   1:L PR[91] 10mm/sec CNT100;
   1:  PR[GP1:91,1] = PR[GP1:90,1] + -19.480;
   1:  PR[GP1:91,2] = PR[GP1:90,2] + 30.902;
   1:L PR[91] 10mm/sec CNT100;
   1:  PR[GP1:91,1] = PR[GP1:90,1] + -27.630;
   1:  PR[GP1:91,2] = PR[GP1:90,2] + 34.001;
   1:L PR[91] 10mm/sec CNT100;
   1:  PR[GP1:91,1] = PR[GP1:90,1] + -29.966;
   1:  PR[GP1:91,2] = PR[GP1:90,2] + 34.343;
   1:L PR[91] 10mm/sec CNT100;
   1:  PR[GP1:91,1] = PR[GP1:90,1] + -37.896;
   1:  PR[GP1:91,2] = PR[GP1:90,2] + 34.907;
   1:L PR[91] 10mm/sec CNT100;
   1:  PR[GP1:91,1] = PR[GP1:90,1] + -42.869;
   1:  PR[GP1:91,2] = PR[GP1:90,2] + 34.106;
   1:L PR[91] 10mm/sec CNT100;
   1:  PR[GP1:91,1] = PR[GP1:90,1] + -48.250;
   1:  PR[GP1:91,2] = PR[GP1:90,2] + 32.901;
   1:L PR[91] 10mm/sec CNT100;
   1:  PR[GP1:91,1] = PR[GP1:90,1] + -54.688;
   1:  PR[GP1:91,2] = PR[GP1:90,2] + 29.663;
   1:L PR[91] 10mm/sec CNT100;
   1:  PR[GP1:91,1] = PR[GP1:90,1] + -57.745;
   1:  PR[GP1:91,2] = PR[GP1:90,2] + 27.940;
   1:L PR[91] 10mm/sec CNT100;
   1:  PR[GP1:91,1] = PR[GP1:90,1] + -63.977;
   1:  PR[GP1:91,2] = PR[GP1:90,2] + 21.826;
   1:L PR[91] 10mm/sec CNT100;
   1:  PR[GP1:91,1] = PR[GP1:90,1] + -65.405;
   1:  PR[GP1:91,2] = PR[GP1:90,2] + 20.322;
   1:L PR[91] 10mm/sec CNT100;
   1:  PR[GP1:91,1] = PR[GP1:90,1] + -69.842;
   1:  PR[GP1:91,2] = PR[GP1:90,2] + 11.800;
   1:L PR[91] 10mm/sec CNT100;
   1:  PR[GP1:91,1] = PR[GP1:90,1] + -70.385;
   1:  PR[GP1:91,2] = PR[GP1:90,2] + 10.702;
   1:L PR[91] 10mm/sec CNT100;
   1:  PR[GP1:91,1] = PR[GP1:90,1] + -71.982;
   1:  PR[GP1:91,2] = PR[GP1:90,2] + 0.854;
   1:L PR[91] 10mm/sec CNT100;
   1:  PR[GP1:91,1] = PR[GP1:90,1] + -72.151;
   1:  PR[GP1:91,2] = PR[GP1:90,2] + -0.013;
   1:L PR[91] 10mm/sec CNT100;
   1:  PR[GP1:91,1] = PR[GP1:90,1] + -70.545;
   1:  PR[GP1:91,2] = PR[GP1:90,2] + -9.656;
   1:L PR[91] 10mm/sec CNT100;
   1:  PR[GP1:91,1] = PR[GP1:90,1] + -70.383;
   1:  PR[GP1:91,2] = PR[GP1:90,2] + -10.713;
   1:L PR[91] 10mm/sec CNT100;
   1:  PR[GP1:91,1] = PR[GP1:90,1] + -69.842;
   1:  PR[GP1:91,2] = PR[GP1:90,2] + -11.809;
   1:L PR[91] 10mm/sec CNT100;
   1:  PR[GP1:91,1] = PR[GP1:90,1] + -65.405;
   1:  PR[GP1:91,2] = PR[GP1:90,2] + -20.330;
   1:L PR[91] 10mm/sec CNT100;
   1:  PR[GP1:91,1] = PR[GP1:90,1] + -63.977;
   1:  PR[GP1:91,2] = PR[GP1:90,2] + -21.835;
   1:L PR[91] 10mm/sec CNT100;
   1:  PR[GP1:91,1] = PR[GP1:90,1] + -57.745;
   1:  PR[GP1:91,2] = PR[GP1:90,2] + -27.949;
   1:L PR[91] 10mm/sec CNT100;
   1:  PR[GP1:91,1] = PR[GP1:90,1] + -54.688;
   1:  PR[GP1:91,2] = PR[GP1:90,2] + -29.672;
   1:L PR[91] 10mm/sec CNT100;
   1:  PR[GP1:91,1] = PR[GP1:90,1] + -48.250;
   1:  PR[GP1:91,2] = PR[GP1:90,2] + -32.910;
   1:L PR[91] 10mm/sec CNT100;
   1:  PR[GP1:91,1] = PR[GP1:90,1] + -42.869;
   1:  PR[GP1:91,2] = PR[GP1:90,2] + -34.115;
   1:L PR[91] 10mm/sec CNT100;
   1:  PR[GP1:91,1] = PR[GP1:90,1] + -37.896;
   1:  PR[GP1:91,2] = PR[GP1:90,2] + -34.916;
   1:L PR[91] 10mm/sec CNT100;
   1:  PR[GP1:91,1] = PR[GP1:90,1] + -29.966;
   1:  PR[GP1:91,2] = PR[GP1:90,2] + -34.352;
   1:L PR[91] 10mm/sec CNT100;
   1:  PR[GP1:91,1] = PR[GP1:90,1] + -27.630;
   1:  PR[GP1:91,2] = PR[GP1:90,2] + -34.009;
   1:L PR[91] 10mm/sec CNT100;
   1:  PR[GP1:91,1] = PR[GP1:90,1] + -19.480;
   1:  PR[GP1:91,2] = PR[GP1:90,2] + -30.911;
   1:L PR[91] 10mm/sec CNT100;
   1:  PR[GP1:91,1] = PR[GP1:90,1] + -18.119;
   1:  PR[GP1:91,2] = PR[GP1:90,2] + -30.431;
   1:L PR[91] 10mm/sec CNT100;
   1:  PR[GP1:91,1] = PR[GP1:90,1] + -17.970;
   1:  PR[GP1:91,2] = PR[GP1:90,2] + -30.350;
   1:L PR[91] 10mm/sec CNT100;
   1:  PR[GP1:91,1] = PR[GP1:90,1] + -10.591;
   1:  PR[GP1:91,2] = PR[GP1:90,2] + -24.946;
   1:L PR[91] 10mm/sec CNT100;
   1:  PR[GP1:91,1] = PR[GP1:90,1] + -9.471;
   1:  PR[GP1:91,2] = PR[GP1:90,2] + -24.053;
   1:L PR[91] 10mm/sec CNT100;
   1:  PR[GP1:91,1] = PR[GP1:90,1] + -8.184;
   1:  PR[GP1:91,2] = PR[GP1:90,2] + -22.548;
   1:L PR[91] 10mm/sec CNT100;
   1:  PR[GP1:91,1] = PR[GP1:90,1] + -4.096;
   1:  PR[GP1:91,2] = PR[GP1:90,2] + -16.957;
   1:L PR[91] 10mm/sec CNT100;
   1:  PR[GP1:91,1] = PR[GP1:90,1] + -2.895;
   1:  PR[GP1:91,2] = PR[GP1:90,2] + -15.610;
   1:L PR[91] 10mm/sec CNT100;
   1:  PR[GP1:91,1] = PR[GP1:90,1] + -0.647;
   1:  PR[GP1:91,2] = PR[GP1:90,2] + -14.295;
   1:L PR[91] 10mm/sec CNT100;
   1:  PR[GP1:91,1] = PR[GP1:90,1] + 1.549;
   1:  PR[GP1:91,2] = PR[GP1:90,2] + -14.273;
   1:L PR[91] 10mm/sec CNT100;
   1:  PR[GP1:91,1] = PR[GP1:90,1] + 2.672;
   1:  PR[GP1:91,2] = PR[GP1:90,2] + -15.619;
   1:L PR[91] 10mm/sec CNT100;
   1:  PR[GP1:91,1] = PR[GP1:90,1] + 3.279;
   1:  PR[GP1:91,2] = PR[GP1:90,2] + -16.002;
   1:L PR[91] 10mm/sec CNT100;
   1:  PR[GP1:91,1] = PR[GP1:90,1] + 4.858;
   1:  PR[GP1:91,2] = PR[GP1:90,2] + -16.866;
   1:L PR[91] 10mm/sec CNT100;
   1:  PR[GP1:91,1] = PR[GP1:90,1] + 9.010;
   1:  PR[GP1:91,2] = PR[GP1:90,2] + -22.547;
   1:L PR[91] 10mm/sec CNT100;
   1:  PR[GP1:91,1] = PR[GP1:90,1] + 10.298;
   1:  PR[GP1:91,2] = PR[GP1:90,2] + -24.056;
   1:L PR[91] 10mm/sec CNT100;
   1:  PR[GP1:91,1] = PR[GP1:90,1] + 18.793;
   1:  PR[GP1:91,2] = PR[GP1:90,2] + -30.355;
   1:L PR[91] 10mm/sec CNT100;
   1:  PR[GP1:91,1] = PR[GP1:90,1] + 18.939;
   1:  PR[GP1:91,2] = PR[GP1:90,2] + -30.434;
   1:L PR[91] 10mm/sec CNT100;
   1:  PR[GP1:91,1] = PR[GP1:90,1] + 20.300;
   1:  PR[GP1:91,2] = PR[GP1:90,2] + -30.914;
   1:L PR[91] 10mm/sec CNT100;
   1:  PR[GP1:91,1] = PR[GP1:90,1] + 28.448;
   1:  PR[GP1:91,2] = PR[GP1:90,2] + -34.007;
   1:L PR[91] 10mm/sec CNT100;
   1:  PR[GP1:91,1] = PR[GP1:90,1] + 30.784;
   1:  PR[GP1:91,2] = PR[GP1:90,2] + -34.351;
   1:L PR[91] 10mm/sec CNT100;
   1:  PR[GP1:91,1] = PR[GP1:90,1] + 38.713;
   1:  PR[GP1:91,2] = PR[GP1:90,2] + -34.916;
   1:L PR[91] 10mm/sec CNT100;
   1:  PR[GP1:91,1] = PR[GP1:90,1] + 43.685;
   1:  PR[GP1:91,2] = PR[GP1:90,2] + -34.116;
   1:L PR[91] 10mm/sec CNT100;
   1:  PR[GP1:91,1] = PR[GP1:90,1] + 49.066;
   1:  PR[GP1:91,2] = PR[GP1:90,2] + -32.909;
   1:L PR[91] 10mm/sec CNT100;
   1:  PR[GP1:91,1] = PR[GP1:90,1] + 55.505;
   1:  PR[GP1:91,2] = PR[GP1:90,2] + -29.676;
   1:L PR[91] 10mm/sec CNT100;
   1:  PR[GP1:91,1] = PR[GP1:90,1] + 58.561;
   1:  PR[GP1:91,2] = PR[GP1:90,2] + -27.956;
   1:L PR[91] 10mm/sec CNT100;
   1:  PR[GP1:91,1] = PR[GP1:90,1] + 64.794;
   1:  PR[GP1:91,2] = PR[GP1:90,2] + -21.832;
   1:L PR[91] 10mm/sec CNT100;
   1:  PR[GP1:91,1] = PR[GP1:90,1] + 66.223;
   1:  PR[GP1:91,2] = PR[GP1:90,2] + -20.323;
   1:L PR[91] 10mm/sec CNT100;
   1:  PR[GP1:91,1] = PR[GP1:90,1] + 70.662;
   1:  PR[GP1:91,2] = PR[GP1:90,2] + -11.822;
   1:L PR[91] 10mm/sec CNT100;
   1:  PR[GP1:91,1] = PR[GP1:90,1] + 71.204;
   1:  PR[GP1:91,2] = PR[GP1:90,2] + -10.730;
   1:L PR[91] 10mm/sec CNT100;
   1:  PR[GP1:91,1] = PR[GP1:90,1] + 72.802;
   1:  PR[GP1:91,2] = PR[GP1:90,2] + -0.866;
   1:L PR[91] 10mm/sec CNT100;
   1:  PR[GP1:91,1] = PR[GP1:90,1] + 72.972;
   1:  PR[GP1:91,2] = PR[GP1:90,2] + 0.004;
   1:L PR[91] 10mm/sec CNT100;
   1:  PR[GP1:91,1] = PR[GP1:90,1] + 71.365;
   1:  PR[GP1:91,2] = PR[GP1:90,2] + 9.663;
   1:L PR[91] 10mm/sec CNT100;
   1:  PR[GP1:91,1] = PR[GP1:90,1] + 71.203;
   1:  PR[GP1:91,2] = PR[GP1:90,2] + 10.724;
   1:L PR[91] 10mm/sec CNT100;
   1:  PR[GP1:91,1] = PR[GP1:90,1] + 70.662;
   1:  PR[GP1:91,2] = PR[GP1:90,2] + 11.813;
   1:L PR[91] 10mm/sec CNT100;
   1:  PR[GP1:91,1] = PR[GP1:90,1] + 66.223;
   1:  PR[GP1:91,2] = PR[GP1:90,2] + 20.314;
   1:L PR[91] 10mm/sec CNT100;
   1:  PR[GP1:91,1] = PR[GP1:90,1] + 64.794;
   1:  PR[GP1:91,2] = PR[GP1:90,2] + 21.823;
   1:L PR[91] 10mm/sec CNT100;
   1:  PR[GP1:91,1] = PR[GP1:90,1] + 58.561;
   1:  PR[GP1:91,2] = PR[GP1:90,2] + 27.947;
   1:L PR[91] 10mm/sec CNT100;
   1:  PR[GP1:91,1] = PR[GP1:90,1] + 55.505;
   1:  PR[GP1:91,2] = PR[GP1:90,2] + 29.667;
   1:L PR[91] 10mm/sec CNT100;
   1:  PR[GP1:91,1] = PR[GP1:90,1] + 49.066;
   1:  PR[GP1:91,2] = PR[GP1:90,2] + 32.900;
   1:L PR[91] 10mm/sec CNT100;
   1:  PR[GP1:91,1] = PR[GP1:90,1] + 43.685;
   1:  PR[GP1:91,2] = PR[GP1:90,2] + 34.107;
   1:L PR[91] 10mm/sec CNT100;
   1:  PR[GP1:91,1] = PR[GP1:90,1] + 38.713;
   1:  PR[GP1:91,2] = PR[GP1:90,2] + 34.908;
   1:L PR[91] 10mm/sec CNT100;
   1:  PR[GP1:91,1] = PR[GP1:90,1] + 30.784;
   1:  PR[GP1:91,2] = PR[GP1:90,2] + 34.342;
   1:L PR[91] 10mm/sec CNT100;
   1:  PR[GP1:91,1] = PR[GP1:90,1] + 28.449;
   1:  PR[GP1:91,2] = PR[GP1:90,2] + 33.998;
   1:L PR[91] 10mm/sec CNT100;
   1:  PR[GP1:91,1] = PR[GP1:90,1] + 20.300;
   1:  PR[GP1:91,2] = PR[GP1:90,2] + 30.905;
   1:L PR[91] 10mm/sec CNT100;
   1:  PR[GP1:91,1] = PR[GP1:90,1] + 18.939;
   1:  PR[GP1:91,2] = PR[GP1:90,2] + 30.426;
   1:L PR[91] 10mm/sec CNT100;
   1:  PR[GP1:91,1] = PR[GP1:90,1] + 18.792;
   1:  PR[GP1:91,2] = PR[GP1:90,2] + 30.346;
   1:L PR[91] 10mm/sec CNT100;
   1:  PR[GP1:91,1] = PR[GP1:90,1] + 11.416;
   1:  PR[GP1:91,2] = PR[GP1:90,2] + 24.939;
   1:L PR[91] 10mm/sec CNT100;
   1:  PR[GP1:91,1] = PR[GP1:90,1] + 10.305;
   1:  PR[GP1:91,2] = PR[GP1:90,2] + 24.055;
   1:L PR[91] 10mm/sec CNT100;
   1:  PR[GP1:91,1] = PR[GP1:90,1] + 9.010;
   1:  PR[GP1:91,2] = PR[GP1:90,2] + 22.538;
   1:L PR[91] 10mm/sec CNT100;
   1:  PR[GP1:91,1] = PR[GP1:90,1] + 4.919;
   1:  PR[GP1:91,2] = PR[GP1:90,2] + 16.940;
   1:L PR[91] 10mm/sec CNT100;
   1:  PR[GP1:91,1] = PR[GP1:90,1] + 3.683;
   1:  PR[GP1:91,2] = PR[GP1:90,2] + 15.580;
   1:L PR[91] 10mm/sec CNT100;
   1:  PR[GP1:91,1] = PR[GP1:90,1] + 1.430;
   1:  PR[GP1:91,2] = PR[GP1:90,2] + 14.266;
   1:L PR[91] 10mm/sec CNT100;
   1:  PR[GP1:91,1] = PR[GP1:90,1] + -0.421;
   1:  PR[GP1:91,2] = PR[GP1:90,2] + 15.206;
   1:  PR[GP1:91,3] = PR[GP1:90,3] + 34.580;
   1:L PR[91] 10mm/sec CNT100;
   1:  PR[GP1:91,1] = PR[GP1:90,1] + -3.157;
   1:  PR[GP1:91,2] = PR[GP1:90,2] + 16.806;
   1:L PR[91] 10mm/sec CNT100;
   1:  PR[GP1:91,1] = PR[GP1:90,1] + -4.121;
   1:  PR[GP1:91,2] = PR[GP1:90,2] + 17.846;
   1:L PR[91] 10mm/sec CNT100;
   1:  PR[GP1:91,1] = PR[GP1:90,1] + -4.130;
   1:  PR[GP1:91,2] = PR[GP1:90,2] + 17.922;
   1:L PR[91] 10mm/sec CNT100;
   1:  PR[GP1:91,1] = PR[GP1:90,1] + -6.847;
   1:  PR[GP1:91,2] = PR[GP1:90,2] + 21.638;
   1:L PR[91] 10mm/sec CNT100;
   1:  PR[GP1:91,1] = PR[GP1:90,1] + -9.039;
   1:  PR[GP1:91,2] = PR[GP1:90,2] + 24.202;
   1:L PR[91] 10mm/sec CNT100;
   1:  PR[GP1:91,1] = PR[GP1:90,1] + -15.244;
   1:  PR[GP1:91,2] = PR[GP1:90,2] + 28.793;
   1:L PR[91] 10mm/sec CNT100;
   1:  PR[GP1:91,1] = PR[GP1:90,1] + -16.880;
   1:  PR[GP1:91,2] = PR[GP1:90,2] + 30.070;
   1:L PR[91] 10mm/sec CNT100;
   1:  PR[GP1:91,1] = PR[GP1:90,1] + -18.082;
   1:  PR[GP1:91,2] = PR[GP1:90,2] + 30.725;
   1:L PR[91] 10mm/sec CNT100;
   1:  PR[GP1:91,1] = PR[GP1:90,1] + -26.011;
   1:  PR[GP1:91,2] = PR[GP1:90,2] + 33.521;
   1:L PR[91] 10mm/sec CNT100;
   1:  PR[GP1:91,1] = PR[GP1:90,1] + -27.773;
   1:  PR[GP1:91,2] = PR[GP1:90,2] + 34.191;
   1:L PR[91] 10mm/sec CNT100;
   1:  PR[GP1:91,1] = PR[GP1:90,1] + -28.222;
   1:  PR[GP1:91,2] = PR[GP1:90,2] + 34.257;
   1:L PR[91] 10mm/sec CNT100;
   1:  PR[GP1:91,1] = PR[GP1:90,1] + -37.971;
   1:  PR[GP1:91,2] = PR[GP1:90,2] + 34.950;
   1:L PR[91] 10mm/sec CNT100;
   1:  PR[GP1:91,1] = PR[GP1:90,1] + -41.193;
   1:  PR[GP1:91,2] = PR[GP1:90,2] + 34.431;
   1:L PR[91] 10mm/sec CNT100;
   1:  PR[GP1:91,1] = PR[GP1:90,1] + -48.233;
   1:  PR[GP1:91,2] = PR[GP1:90,2] + 32.854;
   1:L PR[91] 10mm/sec CNT100;
   1:  PR[GP1:91,1] = PR[GP1:90,1] + -53.210;
   1:  PR[GP1:91,2] = PR[GP1:90,2] + 30.351;
   1:L PR[91] 10mm/sec CNT100;
   1:  PR[GP1:91,1] = PR[GP1:90,1] + -57.636;
   1:  PR[GP1:91,2] = PR[GP1:90,2] + 27.856;
   1:L PR[91] 10mm/sec CNT100;
   1:  PR[GP1:91,1] = PR[GP1:90,1] + -62.792;
   1:  PR[GP1:91,2] = PR[GP1:90,2] + 22.797;
   1:L PR[91] 10mm/sec CNT100;
   1:  PR[GP1:91,1] = PR[GP1:90,1] + -65.219;
   1:  PR[GP1:91,2] = PR[GP1:90,2] + 20.241;
   1:L PR[91] 10mm/sec CNT100;
   1:  PR[GP1:91,1] = PR[GP1:90,1] + -69.012;
   1:  PR[GP1:91,2] = PR[GP1:90,2] + 12.957;
   1:L PR[91] 10mm/sec CNT100;
   1:  PR[GP1:91,1] = PR[GP1:90,1] + -70.148;
   1:  PR[GP1:91,2] = PR[GP1:90,2] + 10.656;
   1:L PR[91] 10mm/sec CNT100;
   1:  PR[GP1:91,1] = PR[GP1:90,1] + -71.535;
   1:  PR[GP1:91,2] = PR[GP1:90,2] + 2.107;
   1:L PR[91] 10mm/sec CNT100;
   1:  PR[GP1:91,1] = PR[GP1:90,1] + -71.700;
   1:  PR[GP1:91,2] = PR[GP1:90,2] + 1.264;
   1:L PR[91] 10mm/sec CNT100;
   1:  PR[GP1:91,1] = PR[GP1:90,1] + -71.894;
   1:  PR[GP1:91,2] = PR[GP1:90,2] + -0.000;
   1:L PR[91] 10mm/sec CNT100;
   1:  PR[GP1:91,1] = PR[GP1:90,1] + -70.486;
   1:  PR[GP1:91,2] = PR[GP1:90,2] + -8.446;
   1:L PR[91] 10mm/sec CNT100;
   1:  PR[GP1:91,1] = PR[GP1:90,1] + -70.147;
   1:  PR[GP1:91,2] = PR[GP1:90,2] + -10.668;
   1:L PR[91] 10mm/sec CNT100;
   1:  PR[GP1:91,1] = PR[GP1:90,1] + -69.012;
   1:  PR[GP1:91,2] = PR[GP1:90,2] + -12.966;
   1:L PR[91] 10mm/sec CNT100;
   1:  PR[GP1:91,1] = PR[GP1:90,1] + -65.219;
   1:  PR[GP1:91,2] = PR[GP1:90,2] + -20.250;
   1:L PR[91] 10mm/sec CNT100;
   1:  PR[GP1:91,1] = PR[GP1:90,1] + -62.792;
   1:  PR[GP1:91,2] = PR[GP1:90,2] + -22.806;
   1:L PR[91] 10mm/sec CNT100;
   1:  PR[GP1:91,1] = PR[GP1:90,1] + -57.636;
   1:  PR[GP1:91,2] = PR[GP1:90,2] + -27.865;
   1:L PR[91] 10mm/sec CNT100;
   1:  PR[GP1:91,1] = PR[GP1:90,1] + -53.210;
   1:  PR[GP1:91,2] = PR[GP1:90,2] + -30.360;
   1:L PR[91] 10mm/sec CNT100;
   1:  PR[GP1:91,1] = PR[GP1:90,1] + -48.233;
   1:  PR[GP1:91,2] = PR[GP1:90,2] + -32.863;
   1:L PR[91] 10mm/sec CNT100;
   1:  PR[GP1:91,1] = PR[GP1:90,1] + -41.193;
   1:  PR[GP1:91,2] = PR[GP1:90,2] + -34.440;
   1:L PR[91] 10mm/sec CNT100;
   1:  PR[GP1:91,1] = PR[GP1:90,1] + -37.971;
   1:  PR[GP1:91,2] = PR[GP1:90,2] + -34.959;
   1:L PR[91] 10mm/sec CNT100;
   1:  PR[GP1:91,1] = PR[GP1:90,1] + -28.222;
   1:  PR[GP1:91,2] = PR[GP1:90,2] + -34.265;
   1:L PR[91] 10mm/sec CNT100;
   1:  PR[GP1:91,1] = PR[GP1:90,1] + -27.773;
   1:  PR[GP1:91,2] = PR[GP1:90,2] + -34.200;
   1:L PR[91] 10mm/sec CNT100;
   1:  PR[GP1:91,1] = PR[GP1:90,1] + -26.012;
   1:  PR[GP1:91,2] = PR[GP1:90,2] + -33.530;
   1:L PR[91] 10mm/sec CNT100;
   1:  PR[GP1:91,1] = PR[GP1:90,1] + -18.991;
   1:  PR[GP1:91,2] = PR[GP1:90,2] + -31.018;
   1:L PR[91] 10mm/sec CNT100;
   1:  PR[GP1:91,1] = PR[GP1:90,1] + -18.073;
   1:  PR[GP1:91,2] = PR[GP1:90,2] + -30.729;
   1:L PR[91] 10mm/sec CNT100;
   1:  PR[GP1:91,1] = PR[GP1:90,1] + -16.871;
   1:  PR[GP1:91,2] = PR[GP1:90,2] + -30.074;
   1:L PR[91] 10mm/sec CNT100;
   1:  PR[GP1:91,1] = PR[GP1:90,1] + -10.967;
   1:  PR[GP1:91,2] = PR[GP1:90,2] + -25.750;
   1:L PR[91] 10mm/sec CNT100;
   1:  PR[GP1:91,1] = PR[GP1:90,1] + -9.046;
   1:  PR[GP1:91,2] = PR[GP1:90,2] + -24.219;
   1:L PR[91] 10mm/sec CNT100;
   1:  PR[GP1:91,1] = PR[GP1:90,1] + -6.847;
   1:  PR[GP1:91,2] = PR[GP1:90,2] + -21.647;
   1:L PR[91] 10mm/sec CNT100;
   1:  PR[GP1:91,1] = PR[GP1:90,1] + -4.019;
   1:  PR[GP1:91,2] = PR[GP1:90,2] + -17.779;
   1:L PR[91] 10mm/sec CNT100;
   1:  PR[GP1:91,1] = PR[GP1:90,1] + -3.163;
   1:  PR[GP1:91,2] = PR[GP1:90,2] + -16.818;
   1:L PR[91] 10mm/sec CNT100;
   1:  PR[GP1:91,1] = PR[GP1:90,1] + -0.421;
   1:  PR[GP1:91,2] = PR[GP1:90,2] + -15.214;
   1:L PR[91] 10mm/sec CNT100;
   1:  PR[GP1:91,1] = PR[GP1:90,1] + 1.334;
   1:  PR[GP1:91,2] = PR[GP1:90,2] + -15.197;
   1:L PR[91] 10mm/sec CNT100;
   1:  PR[GP1:91,1] = PR[GP1:90,1] + 2.206;
   1:  PR[GP1:91,2] = PR[GP1:90,2] + -16.241;
   1:L PR[91] 10mm/sec CNT100;
   1:  PR[GP1:91,1] = PR[GP1:90,1] + 2.636;
   1:  PR[GP1:91,2] = PR[GP1:90,2] + -16.512;
   1:L PR[91] 10mm/sec CNT100;
   1:  PR[GP1:91,1] = PR[GP1:90,1] + 4.784;
   1:  PR[GP1:91,2] = PR[GP1:90,2] + -17.689;
   1:L PR[91] 10mm/sec CNT100;
   1:  PR[GP1:91,1] = PR[GP1:90,1] + 7.677;
   1:  PR[GP1:91,2] = PR[GP1:90,2] + -21.647;
   1:L PR[91] 10mm/sec CNT100;
   1:  PR[GP1:91,1] = PR[GP1:90,1] + 9.883;
   1:  PR[GP1:91,2] = PR[GP1:90,2] + -24.231;
   1:L PR[91] 10mm/sec CNT100;
   1:  PR[GP1:91,1] = PR[GP1:90,1] + 16.085;
   1:  PR[GP1:91,2] = PR[GP1:90,2] + -28.822;
   1:L PR[91] 10mm/sec CNT100;
   1:  PR[GP1:91,1] = PR[GP1:90,1] + 17.705;
   1:  PR[GP1:91,2] = PR[GP1:90,2] + -30.086;
   1:L PR[91] 10mm/sec CNT100;
   1:  PR[GP1:91,1] = PR[GP1:90,1] + 18.899;
   1:  PR[GP1:91,2] = PR[GP1:90,2] + -30.736;
   1:L PR[91] 10mm/sec CNT100;
   1:  PR[GP1:91,1] = PR[GP1:90,1] + 26.831;
   1:  PR[GP1:91,2] = PR[GP1:90,2] + -33.529;
   1:L PR[91] 10mm/sec CNT100;
   1:  PR[GP1:91,1] = PR[GP1:90,1] + 28.593;
   1:  PR[GP1:91,2] = PR[GP1:90,2] + -34.198;
   1:L PR[91] 10mm/sec CNT100;
   1:  PR[GP1:91,1] = PR[GP1:90,1] + 29.043;
   1:  PR[GP1:91,2] = PR[GP1:90,2] + -34.264;
   1:L PR[91] 10mm/sec CNT100;
   1:  PR[GP1:91,1] = PR[GP1:90,1] + 38.789;
   1:  PR[GP1:91,2] = PR[GP1:90,2] + -34.959;
   1:L PR[91] 10mm/sec CNT100;
   1:  PR[GP1:91,1] = PR[GP1:90,1] + 42.011;
   1:  PR[GP1:91,2] = PR[GP1:90,2] + -34.440;
   1:L PR[91] 10mm/sec CNT100;
   1:  PR[GP1:91,1] = PR[GP1:90,1] + 49.050;
   1:  PR[GP1:91,2] = PR[GP1:90,2] + -32.861;
   1:L PR[91] 10mm/sec CNT100;
   1:  PR[GP1:91,1] = PR[GP1:90,1] + 54.028;
   1:  PR[GP1:91,2] = PR[GP1:90,2] + -30.362;
   1:L PR[91] 10mm/sec CNT100;
   1:  PR[GP1:91,1] = PR[GP1:90,1] + 58.453;
   1:  PR[GP1:91,2] = PR[GP1:90,2] + -27.872;
   1:L PR[91] 10mm/sec CNT100;
   1:  PR[GP1:91,1] = PR[GP1:90,1] + 63.610;
   1:  PR[GP1:91,2] = PR[GP1:90,2] + -22.805;
   1:L PR[91] 10mm/sec CNT100;
   1:  PR[GP1:91,1] = PR[GP1:90,1] + 66.038;
   1:  PR[GP1:91,2] = PR[GP1:90,2] + -20.241;
   1:L PR[91] 10mm/sec CNT100;
   1:  PR[GP1:91,1] = PR[GP1:90,1] + 69.832;
   1:  PR[GP1:91,2] = PR[GP1:90,2] + -12.975;
   1:L PR[91] 10mm/sec CNT100;
   1:  PR[GP1:91,1] = PR[GP1:90,1] + 70.969;
   1:  PR[GP1:91,2] = PR[GP1:90,2] + -10.685;
   1:L PR[91] 10mm/sec CNT100;
   1:  PR[GP1:91,1] = PR[GP1:90,1] + 72.356;
   1:  PR[GP1:91,2] = PR[GP1:90,2] + -2.122;
   1:L PR[91] 10mm/sec CNT100;
   1:  PR[GP1:91,1] = PR[GP1:90,1] + 72.521;
   1:  PR[GP1:91,2] = PR[GP1:90,2] + -1.277;
   1:L PR[91] 10mm/sec CNT100;
   1:  PR[GP1:91,1] = PR[GP1:90,1] + 72.715;
   1:  PR[GP1:91,2] = PR[GP1:90,2] + -0.008;
   1:L PR[91] 10mm/sec CNT100;
   1:  PR[GP1:91,1] = PR[GP1:90,1] + 71.306;
   1:  PR[GP1:91,2] = PR[GP1:90,2] + 8.452;
   1:L PR[91] 10mm/sec CNT100;
   1:  PR[GP1:91,1] = PR[GP1:90,1] + 70.967;
   1:  PR[GP1:91,2] = PR[GP1:90,2] + 10.679;
   1:L PR[91] 10mm/sec CNT100;
   1:  PR[GP1:91,1] = PR[GP1:90,1] + 69.832;
   1:  PR[GP1:91,2] = PR[GP1:90,2] + 12.966;
   1:L PR[91] 10mm/sec CNT100;
   1:  PR[GP1:91,1] = PR[GP1:90,1] + 66.038;
   1:  PR[GP1:91,2] = PR[GP1:90,2] + 20.232;
   1:L PR[91] 10mm/sec CNT100;
   1:  PR[GP1:91,1] = PR[GP1:90,1] + 63.610;
   1:  PR[GP1:91,2] = PR[GP1:90,2] + 22.796;
   1:L PR[91] 10mm/sec CNT100;
   1:  PR[GP1:91,1] = PR[GP1:90,1] + 58.453;
   1:  PR[GP1:91,2] = PR[GP1:90,2] + 27.863;
   1:L PR[91] 10mm/sec CNT100;
   1:  PR[GP1:91,1] = PR[GP1:90,1] + 54.028;
   1:  PR[GP1:91,2] = PR[GP1:90,2] + 30.353;
   1:L PR[91] 10mm/sec CNT100;
   1:  PR[GP1:91,1] = PR[GP1:90,1] + 49.050;
   1:  PR[GP1:91,2] = PR[GP1:90,2] + 32.853;
   1:L PR[91] 10mm/sec CNT100;
   1:  PR[GP1:91,1] = PR[GP1:90,1] + 42.011;
   1:  PR[GP1:91,2] = PR[GP1:90,2] + 34.432;
   1:L PR[91] 10mm/sec CNT100;
   1:  PR[GP1:91,1] = PR[GP1:90,1] + 38.789;
   1:  PR[GP1:91,2] = PR[GP1:90,2] + 34.950;
   1:L PR[91] 10mm/sec CNT100;
   1:  PR[GP1:91,1] = PR[GP1:90,1] + 29.043;
   1:  PR[GP1:91,2] = PR[GP1:90,2] + 34.255;
   1:L PR[91] 10mm/sec CNT100;
   1:  PR[GP1:91,1] = PR[GP1:90,1] + 28.593;
   1:  PR[GP1:91,2] = PR[GP1:90,2] + 34.189;
   1:L PR[91] 10mm/sec CNT100;
   1:  PR[GP1:91,1] = PR[GP1:90,1] + 26.833;
   1:  PR[GP1:91,2] = PR[GP1:90,2] + 33.521;
   1:L PR[91] 10mm/sec CNT100;
   1:  PR[GP1:91,1] = PR[GP1:90,1] + 19.811;
   1:  PR[GP1:91,2] = PR[GP1:90,2] + 31.011;
   1:L PR[91] 10mm/sec CNT100;
   1:  PR[GP1:91,1] = PR[GP1:90,1] + 18.890;
   1:  PR[GP1:91,2] = PR[GP1:90,2] + 30.722;
   1:L PR[91] 10mm/sec CNT100;
   1:  PR[GP1:91,1] = PR[GP1:90,1] + 17.698;
   1:  PR[GP1:91,2] = PR[GP1:90,2] + 30.073;
   1:L PR[91] 10mm/sec CNT100;
   1:  PR[GP1:91,1] = PR[GP1:90,1] + 11.794;
   1:  PR[GP1:91,2] = PR[GP1:90,2] + 25.745;
   1:L PR[91] 10mm/sec CNT100;
   1:  PR[GP1:91,1] = PR[GP1:90,1] + 9.889;
   1:  PR[GP1:91,2] = PR[GP1:90,2] + 24.230;
   1:L PR[91] 10mm/sec CNT100;
   1:  PR[GP1:91,1] = PR[GP1:90,1] + 7.677;
   1:  PR[GP1:91,2] = PR[GP1:90,2] + 21.638;
   1:L PR[91] 10mm/sec CNT100;
   1:  PR[GP1:91,1] = PR[GP1:90,1] + 4.845;
   1:  PR[GP1:91,2] = PR[GP1:90,2] + 17.763;
   1:L PR[91] 10mm/sec CNT100;
   1:  PR[GP1:91,1] = PR[GP1:90,1] + 3.964;
   1:  PR[GP1:91,2] = PR[GP1:90,2] + 16.793;
   1:L PR[91] 10mm/sec CNT100;
   1:  PR[GP1:91,1] = PR[GP1:90,1] + 1.216;
   1:  PR[GP1:91,2] = PR[GP1:90,2] + 15.190;
   1:L PR[91] 10mm/sec CNT100;
   1:  PR[GP1:91,1] = PR[GP1:90,1] + -0.195;
   1:  PR[GP1:91,2] = PR[GP1:90,2] + 16.125;
   1:  PR[GP1:91,3] = PR[GP1:90,3] + 35.910;
   1:L PR[91] 10mm/sec CNT100;
   1:  PR[GP1:91,1] = PR[GP1:90,1] + -3.425;
   1:  PR[GP1:91,2] = PR[GP1:90,2] + 18.015;
   1:L PR[91] 10mm/sec CNT100;
   1:  PR[GP1:91,1] = PR[GP1:90,1] + -4.046;
   1:  PR[GP1:91,2] = PR[GP1:90,2] + 18.684;
   1:L PR[91] 10mm/sec CNT100;
   1:  PR[GP1:91,1] = PR[GP1:90,1] + -4.053;
   1:  PR[GP1:91,2] = PR[GP1:90,2] + 18.743;
   1:L PR[91] 10mm/sec CNT100;
   1:  PR[GP1:91,1] = PR[GP1:90,1] + -5.511;
   1:  PR[GP1:91,2] = PR[GP1:90,2] + 20.737;
   1:L PR[91] 10mm/sec CNT100;
   1:  PR[GP1:91,1] = PR[GP1:90,1] + -8.614;
   1:  PR[GP1:91,2] = PR[GP1:90,2] + 24.368;
   1:L PR[91] 10mm/sec CNT100;
   1:  PR[GP1:91,1] = PR[GP1:90,1] + -12.771;
   1:  PR[GP1:91,2] = PR[GP1:90,2] + 27.443;
   1:L PR[91] 10mm/sec CNT100;
   1:  PR[GP1:91,1] = PR[GP1:90,1] + -15.781;
   1:  PR[GP1:91,2] = PR[GP1:90,2] + 29.793;
   1:L PR[91] 10mm/sec CNT100;
   1:  PR[GP1:91,1] = PR[GP1:90,1] + -18.045;
   1:  PR[GP1:91,2] = PR[GP1:90,2] + 31.028;
   1:L PR[91] 10mm/sec CNT100;
   1:  PR[GP1:91,1] = PR[GP1:90,1] + -26.386;
   1:  PR[GP1:91,2] = PR[GP1:90,2] + 33.969;
   1:L PR[91] 10mm/sec CNT100;
   1:  PR[GP1:91,1] = PR[GP1:90,1] + -27.328;
   1:  PR[GP1:91,2] = PR[GP1:90,2] + 34.276;
   1:L PR[91] 10mm/sec CNT100;
   1:  PR[GP1:91,1] = PR[GP1:90,1] + -27.938;
   1:  PR[GP1:91,2] = PR[GP1:90,2] + 34.364;
   1:L PR[91] 10mm/sec CNT100;
   1:  PR[GP1:91,1] = PR[GP1:90,1] + -32.367;
   1:  PR[GP1:91,2] = PR[GP1:90,2] + 34.589;
   1:L PR[91] 10mm/sec CNT100;
   1:  PR[GP1:91,1] = PR[GP1:90,1] + -38.045;
   1:  PR[GP1:91,2] = PR[GP1:90,2] + 34.993;
   1:L PR[91] 10mm/sec CNT100;
   1:  PR[GP1:91,1] = PR[GP1:90,1] + -39.517;
   1:  PR[GP1:91,2] = PR[GP1:90,2] + 34.756;
   1:L PR[91] 10mm/sec CNT100;
   1:  PR[GP1:91,1] = PR[GP1:90,1] + -48.216;
   1:  PR[GP1:91,2] = PR[GP1:90,2] + 32.807;
   1:L PR[91] 10mm/sec CNT100;
   1:  PR[GP1:91,1] = PR[GP1:90,1] + -51.732;
   1:  PR[GP1:91,2] = PR[GP1:90,2] + 31.039;
   1:L PR[91] 10mm/sec CNT100;
   1:  PR[GP1:91,1] = PR[GP1:90,1] + -57.527;
   1:  PR[GP1:91,2] = PR[GP1:90,2] + 27.773;
   1:L PR[91] 10mm/sec CNT100;
   1:  PR[GP1:91,1] = PR[GP1:90,1] + -61.608;
   1:  PR[GP1:91,2] = PR[GP1:90,2] + 23.768;
   1:L PR[91] 10mm/sec CNT100;
   1:  PR[GP1:91,1] = PR[GP1:90,1] + -65.033;
   1:  PR[GP1:91,2] = PR[GP1:90,2] + 20.161;
   1:L PR[91] 10mm/sec CNT100;
   1:  PR[GP1:91,1] = PR[GP1:90,1] + -68.181;
   1:  PR[GP1:91,2] = PR[GP1:90,2] + 14.114;
   1:L PR[91] 10mm/sec CNT100;
   1:  PR[GP1:91,1] = PR[GP1:90,1] + -69.912;
   1:  PR[GP1:91,2] = PR[GP1:90,2] + 10.611;
   1:L PR[91] 10mm/sec CNT100;
   1:  PR[GP1:91,1] = PR[GP1:90,1] + -71.089;
   1:  PR[GP1:91,2] = PR[GP1:90,2] + 3.359;
   1:L PR[91] 10mm/sec CNT100;
   1:  PR[GP1:91,1] = PR[GP1:90,1] + -71.229;
   1:  PR[GP1:91,2] = PR[GP1:90,2] + 2.644;
   1:L PR[91] 10mm/sec CNT100;
   1:  PR[GP1:91,1] = PR[GP1:90,1] + -71.634;
   1:  PR[GP1:91,2] = PR[GP1:90,2] + -0.000;
   1:L PR[91] 10mm/sec CNT100;
   1:  PR[GP1:91,1] = PR[GP1:90,1] + -70.428;
   1:  PR[GP1:91,2] = PR[GP1:90,2] + -7.237;
   1:L PR[91] 10mm/sec CNT100;
   1:  PR[GP1:91,1] = PR[GP1:90,1] + -69.911;
   1:  PR[GP1:91,2] = PR[GP1:90,2] + -10.622;
   1:L PR[91] 10mm/sec CNT100;
   1:  PR[GP1:91,1] = PR[GP1:90,1] + -68.181;
   1:  PR[GP1:91,2] = PR[GP1:90,2] + -14.123;
   1:L PR[91] 10mm/sec CNT100;
   1:  PR[GP1:91,1] = PR[GP1:90,1] + -65.033;
   1:  PR[GP1:91,2] = PR[GP1:90,2] + -20.169;
   1:L PR[91] 10mm/sec CNT100;
   1:  PR[GP1:91,1] = PR[GP1:90,1] + -61.608;
   1:  PR[GP1:91,2] = PR[GP1:90,2] + -23.777;
   1:L PR[91] 10mm/sec CNT100;
   1:  PR[GP1:91,1] = PR[GP1:90,1] + -57.527;
   1:  PR[GP1:91,2] = PR[GP1:90,2] + -27.782;
   1:L PR[91] 10mm/sec CNT100;
   1:  PR[GP1:91,1] = PR[GP1:90,1] + -51.732;
   1:  PR[GP1:91,2] = PR[GP1:90,2] + -31.048;
   1:L PR[91] 10mm/sec CNT100;
   1:  PR[GP1:91,1] = PR[GP1:90,1] + -48.216;
   1:  PR[GP1:91,2] = PR[GP1:90,2] + -32.816;
   1:L PR[91] 10mm/sec CNT100;
   1:  PR[GP1:91,1] = PR[GP1:90,1] + -39.517;
   1:  PR[GP1:91,2] = PR[GP1:90,2] + -34.764;
   1:L PR[91] 10mm/sec CNT100;
   1:  PR[GP1:91,1] = PR[GP1:90,1] + -38.045;
   1:  PR[GP1:91,2] = PR[GP1:90,2] + -35.001;
   1:L PR[91] 10mm/sec CNT100;
   1:  PR[GP1:91,1] = PR[GP1:90,1] + -32.367;
   1:  PR[GP1:91,2] = PR[GP1:90,2] + -34.598;
   1:L PR[91] 10mm/sec CNT100;
   1:  PR[GP1:91,1] = PR[GP1:90,1] + -27.938;
   1:  PR[GP1:91,2] = PR[GP1:90,2] + -34.373;
   1:L PR[91] 10mm/sec CNT100;
   1:  PR[GP1:91,1] = PR[GP1:90,1] + -27.337;
   1:  PR[GP1:91,2] = PR[GP1:90,2] + -34.286;
   1:L PR[91] 10mm/sec CNT100;
   1:  PR[GP1:91,1] = PR[GP1:90,1] + -19.748;
   1:  PR[GP1:91,2] = PR[GP1:90,2] + -31.570;
   1:L PR[91] 10mm/sec CNT100;
   1:  PR[GP1:91,1] = PR[GP1:90,1] + -18.036;
   1:  PR[GP1:91,2] = PR[GP1:90,2] + -31.032;
   1:L PR[91] 10mm/sec CNT100;
   1:  PR[GP1:91,1] = PR[GP1:90,1] + -15.773;
   1:  PR[GP1:91,2] = PR[GP1:90,2] + -29.798;
   1:L PR[91] 10mm/sec CNT100;
   1:  PR[GP1:91,1] = PR[GP1:90,1] + -11.342;
   1:  PR[GP1:91,2] = PR[GP1:90,2] + -26.553;
   1:L PR[91] 10mm/sec CNT100;
   1:  PR[GP1:91,1] = PR[GP1:90,1] + -8.621;
   1:  PR[GP1:91,2] = PR[GP1:90,2] + -24.385;
   1:L PR[91] 10mm/sec CNT100;
   1:  PR[GP1:91,1] = PR[GP1:90,1] + -5.511;
   1:  PR[GP1:91,2] = PR[GP1:90,2] + -20.746;
   1:L PR[91] 10mm/sec CNT100;
   1:  PR[GP1:91,1] = PR[GP1:90,1] + -3.942;
   1:  PR[GP1:91,2] = PR[GP1:90,2] + -18.600;
   1:L PR[91] 10mm/sec CNT100;
   1:  PR[GP1:91,1] = PR[GP1:90,1] + -3.430;
   1:  PR[GP1:91,2] = PR[GP1:90,2] + -18.026;
   1:L PR[91] 10mm/sec CNT100;
   1:  PR[GP1:91,1] = PR[GP1:90,1] + -0.195;
   1:  PR[GP1:91,2] = PR[GP1:90,2] + -16.134;
   1:L PR[91] 10mm/sec CNT100;
   1:  PR[GP1:91,1] = PR[GP1:90,1] + 1.120;
   1:  PR[GP1:91,2] = PR[GP1:90,2] + -16.121;
   1:L PR[91] 10mm/sec CNT100;
   1:  PR[GP1:91,1] = PR[GP1:90,1] + 1.739;
   1:  PR[GP1:91,2] = PR[GP1:90,2] + -16.863;
   1:L PR[91] 10mm/sec CNT100;
   1:  PR[GP1:91,1] = PR[GP1:90,1] + 1.993;
   1:  PR[GP1:91,2] = PR[GP1:90,2] + -17.023;
   1:L PR[91] 10mm/sec CNT100;
   1:  PR[GP1:91,1] = PR[GP1:90,1] + 4.710;
   1:  PR[GP1:91,2] = PR[GP1:90,2] + -18.511;
   1:L PR[91] 10mm/sec CNT100;
   1:  PR[GP1:91,1] = PR[GP1:90,1] + 6.344;
   1:  PR[GP1:91,2] = PR[GP1:90,2] + -20.747;
   1:L PR[91] 10mm/sec CNT100;
   1:  PR[GP1:91,1] = PR[GP1:90,1] + 9.467;
   1:  PR[GP1:91,2] = PR[GP1:90,2] + -24.406;
   1:L PR[91] 10mm/sec CNT100;
   1:  PR[GP1:91,1] = PR[GP1:90,1] + 13.628;
   1:  PR[GP1:91,2] = PR[GP1:90,2] + -27.486;
   1:L PR[91] 10mm/sec CNT100;
   1:  PR[GP1:91,1] = PR[GP1:90,1] + 16.611;
   1:  PR[GP1:91,2] = PR[GP1:90,2] + -29.814;
   1:L PR[91] 10mm/sec CNT100;
   1:  PR[GP1:91,1] = PR[GP1:90,1] + 18.860;
   1:  PR[GP1:91,2] = PR[GP1:90,2] + -31.037;
   1:L PR[91] 10mm/sec CNT100;
   1:  PR[GP1:91,1] = PR[GP1:90,1] + 27.204;
   1:  PR[GP1:91,2] = PR[GP1:90,2] + -33.975;
   1:L PR[91] 10mm/sec CNT100;
   1:  PR[GP1:91,1] = PR[GP1:90,1] + 28.148;
   1:  PR[GP1:91,2] = PR[GP1:90,2] + -34.283;
   1:L PR[91] 10mm/sec CNT100;
   1:  PR[GP1:91,1] = PR[GP1:90,1] + 28.758;
   1:  PR[GP1:91,2] = PR[GP1:90,2] + -34.372;
   1:L PR[91] 10mm/sec CNT100;
   1:  PR[GP1:91,1] = PR[GP1:90,1] + 33.188;
   1:  PR[GP1:91,2] = PR[GP1:90,2] + -34.597;
   1:L PR[91] 10mm/sec CNT100;
   1:  PR[GP1:91,1] = PR[GP1:90,1] + 38.865;
   1:  PR[GP1:91,2] = PR[GP1:90,2] + -35.002;
   1:L PR[91] 10mm/sec CNT100;
   1:  PR[GP1:91,1] = PR[GP1:90,1] + 40.336;
   1:  PR[GP1:91,2] = PR[GP1:90,2] + -34.765;
   1:L PR[91] 10mm/sec CNT100;
   1:  PR[GP1:91,1] = PR[GP1:90,1] + 49.034;
   1:  PR[GP1:91,2] = PR[GP1:90,2] + -32.814;
   1:L PR[91] 10mm/sec CNT100;
   1:  PR[GP1:91,1] = PR[GP1:90,1] + 52.551;
   1:  PR[GP1:91,2] = PR[GP1:90,2] + -31.049;
   1:L PR[91] 10mm/sec CNT100;
   1:  PR[GP1:91,1] = PR[GP1:90,1] + 58.344;
   1:  PR[GP1:91,2] = PR[GP1:90,2] + -27.788;
   1:L PR[91] 10mm/sec CNT100;
   1:  PR[GP1:91,1] = PR[GP1:90,1] + 62.426;
   1:  PR[GP1:91,2] = PR[GP1:90,2] + -23.778;
   1:L PR[91] 10mm/sec CNT100;
   1:  PR[GP1:91,1] = PR[GP1:90,1] + 65.852;
   1:  PR[GP1:91,2] = PR[GP1:90,2] + -20.159;
   1:L PR[91] 10mm/sec CNT100;
   1:  PR[GP1:91,1] = PR[GP1:90,1] + 69.002;
   1:  PR[GP1:91,2] = PR[GP1:90,2] + -14.127;
   1:L PR[91] 10mm/sec CNT100;
   1:  PR[GP1:91,1] = PR[GP1:90,1] + 70.733;
   1:  PR[GP1:91,2] = PR[GP1:90,2] + -10.641;
   1:L PR[91] 10mm/sec CNT100;
   1:  PR[GP1:91,1] = PR[GP1:90,1] + 71.909;
   1:  PR[GP1:91,2] = PR[GP1:90,2] + -3.378;
   1:L PR[91] 10mm/sec CNT100;
   1:  PR[GP1:91,1] = PR[GP1:90,1] + 72.049;
   1:  PR[GP1:91,2] = PR[GP1:90,2] + -2.661;
   1:L PR[91] 10mm/sec CNT100;
   1:  PR[GP1:91,1] = PR[GP1:90,1] + 72.455;
   1:  PR[GP1:91,2] = PR[GP1:90,2] + -0.008;
   1:L PR[91] 10mm/sec CNT100;
   1:  PR[GP1:91,1] = PR[GP1:90,1] + 71.248;
   1:  PR[GP1:91,2] = PR[GP1:90,2] + 7.241;
   1:L PR[91] 10mm/sec CNT100;
   1:  PR[GP1:91,1] = PR[GP1:90,1] + 70.731;
   1:  PR[GP1:91,2] = PR[GP1:90,2] + 10.635;
   1:L PR[91] 10mm/sec CNT100;
   1:  PR[GP1:91,1] = PR[GP1:90,1] + 69.002;
   1:  PR[GP1:91,2] = PR[GP1:90,2] + 14.118;
   1:L PR[91] 10mm/sec CNT100;
   1:  PR[GP1:91,1] = PR[GP1:90,1] + 65.852;
   1:  PR[GP1:91,2] = PR[GP1:90,2] + 20.150;
   1:L PR[91] 10mm/sec CNT100;
   1:  PR[GP1:91,1] = PR[GP1:90,1] + 62.426;
   1:  PR[GP1:91,2] = PR[GP1:90,2] + 23.769;
   1:L PR[91] 10mm/sec CNT100;
   1:  PR[GP1:91,1] = PR[GP1:90,1] + 58.344;
   1:  PR[GP1:91,2] = PR[GP1:90,2] + 27.779;
   1:L PR[91] 10mm/sec CNT100;
   1:  PR[GP1:91,1] = PR[GP1:90,1] + 52.551;
   1:  PR[GP1:91,2] = PR[GP1:90,2] + 31.040;
   1:L PR[91] 10mm/sec CNT100;
   1:  PR[GP1:91,1] = PR[GP1:90,1] + 49.034;
   1:  PR[GP1:91,2] = PR[GP1:90,2] + 32.805;
   1:L PR[91] 10mm/sec CNT100;
   1:  PR[GP1:91,1] = PR[GP1:90,1] + 40.336;
   1:  PR[GP1:91,2] = PR[GP1:90,2] + 34.756;
   1:L PR[91] 10mm/sec CNT100;
   1:  PR[GP1:91,1] = PR[GP1:90,1] + 38.865;
   1:  PR[GP1:91,2] = PR[GP1:90,2] + 34.993;
   1:L PR[91] 10mm/sec CNT100;
   1:  PR[GP1:91,1] = PR[GP1:90,1] + 33.188;
   1:  PR[GP1:91,2] = PR[GP1:90,2] + 34.588;
   1:L PR[91] 10mm/sec CNT100;
   1:  PR[GP1:91,1] = PR[GP1:90,1] + 28.758;
   1:  PR[GP1:91,2] = PR[GP1:90,2] + 34.363;
   1:L PR[91] 10mm/sec CNT100;
   1:  PR[GP1:91,1] = PR[GP1:90,1] + 28.157;
   1:  PR[GP1:91,2] = PR[GP1:90,2] + 34.275;
   1:L PR[91] 10mm/sec CNT100;
   1:  PR[GP1:91,1] = PR[GP1:90,1] + 20.568;
   1:  PR[GP1:91,2] = PR[GP1:90,2] + 31.563;
   1:L PR[91] 10mm/sec CNT100;
   1:  PR[GP1:91,1] = PR[GP1:90,1] + 18.851;
   1:  PR[GP1:91,2] = PR[GP1:90,2] + 31.023;
   1:L PR[91] 10mm/sec CNT100;
   1:  PR[GP1:91,1] = PR[GP1:90,1] + 16.604;
   1:  PR[GP1:91,2] = PR[GP1:90,2] + 29.801;
   1:L PR[91] 10mm/sec CNT100;
   1:  PR[GP1:91,1] = PR[GP1:90,1] + 12.173;
   1:  PR[GP1:91,2] = PR[GP1:90,2] + 26.552;
   1:L PR[91] 10mm/sec CNT100;
   1:  PR[GP1:91,1] = PR[GP1:90,1] + 9.474;
   1:  PR[GP1:91,2] = PR[GP1:90,2] + 24.405;
   1:L PR[91] 10mm/sec CNT100;
   1:  PR[GP1:91,1] = PR[GP1:90,1] + 6.344;
   1:  PR[GP1:91,2] = PR[GP1:90,2] + 20.738;
   1:L PR[91] 10mm/sec CNT100;
   1:  PR[GP1:91,1] = PR[GP1:90,1] + 4.771;
   1:  PR[GP1:91,2] = PR[GP1:90,2] + 18.585;
   1:L PR[91] 10mm/sec CNT100;
   1:  PR[GP1:91,1] = PR[GP1:90,1] + 4.245;
   1:  PR[GP1:91,2] = PR[GP1:90,2] + 18.006;
   1:L PR[91] 10mm/sec CNT100;
   1:  PR[GP1:91,1] = PR[GP1:90,1] + 1.001;
   1:  PR[GP1:91,2] = PR[GP1:90,2] + 16.114;
   1:L PR[91] 10mm/sec CNT100;
   1:  PR[GP1:91,1] = PR[GP1:90,1] + 0.031;
   1:  PR[GP1:91,2] = PR[GP1:90,2] + 17.045;
   1:  PR[GP1:91,3] = PR[GP1:90,3] + 37.240;
   1:L PR[91] 10mm/sec CNT100;
   1:  PR[GP1:91,1] = PR[GP1:90,1] + -3.693;
   1:  PR[GP1:91,2] = PR[GP1:90,2] + 19.223;
   1:L PR[91] 10mm/sec CNT100;
   1:  PR[GP1:91,1] = PR[GP1:90,1] + -3.861;
   1:  PR[GP1:91,2] = PR[GP1:90,2] + 19.404;
   1:L PR[91] 10mm/sec CNT100;
   1:  PR[GP1:91,1] = PR[GP1:90,1] + -4.175;
   1:  PR[GP1:91,2] = PR[GP1:90,2] + 19.837;
   1:L PR[91] 10mm/sec CNT100;
   1:  PR[GP1:91,1] = PR[GP1:90,1] + -8.189;
   1:  PR[GP1:91,2] = PR[GP1:90,2] + 24.534;
   1:L PR[91] 10mm/sec CNT100;
   1:  PR[GP1:91,1] = PR[GP1:90,1] + -10.297;
   1:  PR[GP1:91,2] = PR[GP1:90,2] + 26.093;
   1:L PR[91] 10mm/sec CNT100;
   1:  PR[GP1:91,1] = PR[GP1:90,1] + -14.682;
   1:  PR[GP1:91,2] = PR[GP1:90,2] + 29.517;
   1:L PR[91] 10mm/sec CNT100;
   1:  PR[GP1:91,1] = PR[GP1:90,1] + -18.008;
   1:  PR[GP1:91,2] = PR[GP1:90,2] + 31.331;
   1:L PR[91] 10mm/sec CNT100;
   1:  PR[GP1:91,1] = PR[GP1:90,1] + -24.335;
   1:  PR[GP1:91,2] = PR[GP1:90,2] + 33.562;
   1:L PR[91] 10mm/sec CNT100;
   1:  PR[GP1:91,1] = PR[GP1:90,1] + -26.671;
   1:  PR[GP1:91,2] = PR[GP1:90,2] + 34.322;
   1:L PR[91] 10mm/sec CNT100;
   1:  PR[GP1:91,1] = PR[GP1:90,1] + -28.243;
   1:  PR[GP1:91,2] = PR[GP1:90,2] + 34.550;
   1:L PR[91] 10mm/sec CNT100;
   1:  PR[GP1:91,1] = PR[GP1:90,1] + -38.058;
   1:  PR[GP1:91,2] = PR[GP1:90,2] + 35.038;
   1:L PR[91] 10mm/sec CNT100;
   1:  PR[GP1:91,1] = PR[GP1:90,1] + -48.199;
   1:  PR[GP1:91,2] = PR[GP1:90,2] + 32.761;
   1:L PR[91] 10mm/sec CNT100;
   1:  PR[GP1:91,1] = PR[GP1:90,1] + -50.255;
   1:  PR[GP1:91,2] = PR[GP1:90,2] + 31.727;
   1:L PR[91] 10mm/sec CNT100;
   1:  PR[GP1:91,1] = PR[GP1:90,1] + -57.417;
   1:  PR[GP1:91,2] = PR[GP1:90,2] + 27.689;
   1:L PR[91] 10mm/sec CNT100;
   1:  PR[GP1:91,1] = PR[GP1:90,1] + -60.424;
   1:  PR[GP1:91,2] = PR[GP1:90,2] + 24.740;
   1:L PR[91] 10mm/sec CNT100;
   1:  PR[GP1:91,1] = PR[GP1:90,1] + -64.847;
   1:  PR[GP1:91,2] = PR[GP1:90,2] + 20.080;
   1:L PR[91] 10mm/sec CNT100;
   1:  PR[GP1:91,1] = PR[GP1:90,1] + -67.351;
   1:  PR[GP1:91,2] = PR[GP1:90,2] + 15.272;
   1:L PR[91] 10mm/sec CNT100;
   1:  PR[GP1:91,1] = PR[GP1:90,1] + -69.676;
   1:  PR[GP1:91,2] = PR[GP1:90,2] + 10.565;
   1:L PR[91] 10mm/sec CNT100;
   1:  PR[GP1:91,1] = PR[GP1:90,1] + -70.642;
   1:  PR[GP1:91,2] = PR[GP1:90,2] + 4.611;
   1:L PR[91] 10mm/sec CNT100;
   1:  PR[GP1:91,1] = PR[GP1:90,1] + -70.757;
   1:  PR[GP1:91,2] = PR[GP1:90,2] + 4.023;
   1:L PR[91] 10mm/sec CNT100;
   1:  PR[GP1:91,1] = PR[GP1:90,1] + -71.374;
   1:  PR[GP1:91,2] = PR[GP1:90,2] + -0.000;
   1:L PR[91] 10mm/sec CNT100;
   1:  PR[GP1:91,1] = PR[GP1:90,1] + -70.369;
   1:  PR[GP1:91,2] = PR[GP1:90,2] + -6.028;
   1:L PR[91] 10mm/sec CNT100;
   1:  PR[GP1:91,1] = PR[GP1:90,1] + -69.675;
   1:  PR[GP1:91,2] = PR[GP1:90,2] + -10.577;
   1:L PR[91] 10mm/sec CNT100;
   1:  PR[GP1:91,1] = PR[GP1:90,1] + -67.351;
   1:  PR[GP1:91,2] = PR[GP1:90,2] + -15.280;
   1:L PR[91] 10mm/sec CNT100;
   1:  PR[GP1:91,1] = PR[GP1:90,1] + -64.847;
   1:  PR[GP1:91,2] = PR[GP1:90,2] + -20.089;
   1:L PR[91] 10mm/sec CNT100;
   1:  PR[GP1:91,1] = PR[GP1:90,1] + -60.424;
   1:  PR[GP1:91,2] = PR[GP1:90,2] + -24.749;
   1:L PR[91] 10mm/sec CNT100;
   1:  PR[GP1:91,1] = PR[GP1:90,1] + -57.417;
   1:  PR[GP1:91,2] = PR[GP1:90,2] + -27.698;
   1:L PR[91] 10mm/sec CNT100;
   1:  PR[GP1:91,1] = PR[GP1:90,1] + -50.254;
   1:  PR[GP1:91,2] = PR[GP1:90,2] + -31.736;
   1:L PR[91] 10mm/sec CNT100;
   1:  PR[GP1:91,1] = PR[GP1:90,1] + -48.199;
   1:  PR[GP1:91,2] = PR[GP1:90,2] + -32.769;
   1:L PR[91] 10mm/sec CNT100;
   1:  PR[GP1:91,1] = PR[GP1:90,1] + -38.058;
   1:  PR[GP1:91,2] = PR[GP1:90,2] + -35.047;
   1:L PR[91] 10mm/sec CNT100;
   1:  PR[GP1:91,1] = PR[GP1:90,1] + -28.243;
   1:  PR[GP1:91,2] = PR[GP1:90,2] + -34.559;
   1:L PR[91] 10mm/sec CNT100;
   1:  PR[GP1:91,1] = PR[GP1:90,1] + -26.679;
   1:  PR[GP1:91,2] = PR[GP1:90,2] + -34.332;
   1:L PR[91] 10mm/sec CNT100;
   1:  PR[GP1:91,1] = PR[GP1:90,1] + -20.505;
   1:  PR[GP1:91,2] = PR[GP1:90,2] + -32.123;
   1:L PR[91] 10mm/sec CNT100;
   1:  PR[GP1:91,1] = PR[GP1:90,1] + -17.999;
   1:  PR[GP1:91,2] = PR[GP1:90,2] + -31.335;
   1:L PR[91] 10mm/sec CNT100;
   1:  PR[GP1:91,1] = PR[GP1:90,1] + -14.674;
   1:  PR[GP1:91,2] = PR[GP1:90,2] + -29.522;
   1:L PR[91] 10mm/sec CNT100;
   1:  PR[GP1:91,1] = PR[GP1:90,1] + -11.717;
   1:  PR[GP1:91,2] = PR[GP1:90,2] + -27.356;
   1:L PR[91] 10mm/sec CNT100;
   1:  PR[GP1:91,1] = PR[GP1:90,1] + -8.196;
   1:  PR[GP1:91,2] = PR[GP1:90,2] + -24.551;
   1:L PR[91] 10mm/sec CNT100;
   1:  PR[GP1:91,1] = PR[GP1:90,1] + -4.170;
   1:  PR[GP1:91,2] = PR[GP1:90,2] + -19.840;
   1:L PR[91] 10mm/sec CNT100;
   1:  PR[GP1:91,1] = PR[GP1:90,1] + -3.719;
   1:  PR[GP1:91,2] = PR[GP1:90,2] + -19.247;
   1:L PR[91] 10mm/sec CNT100;
   1:  PR[GP1:91,1] = PR[GP1:90,1] + 0.031;
   1:  PR[GP1:91,2] = PR[GP1:90,2] + -17.054;
   1:L PR[91] 10mm/sec CNT100;
   1:  PR[GP1:91,1] = PR[GP1:90,1] + 0.905;
   1:  PR[GP1:91,2] = PR[GP1:90,2] + -17.045;
   1:L PR[91] 10mm/sec CNT100;
   1:  PR[GP1:91,1] = PR[GP1:90,1] + 1.272;
   1:  PR[GP1:91,2] = PR[GP1:90,2] + -17.485;
   1:L PR[91] 10mm/sec CNT100;
   1:  PR[GP1:91,1] = PR[GP1:90,1] + 1.349;
   1:  PR[GP1:91,2] = PR[GP1:90,2] + -17.534;
   1:L PR[91] 10mm/sec CNT100;
   1:  PR[GP1:91,1] = PR[GP1:90,1] + 4.636;
   1:  PR[GP1:91,2] = PR[GP1:90,2] + -19.334;
   1:L PR[91] 10mm/sec CNT100;
   1:  PR[GP1:91,1] = PR[GP1:90,1] + 5.011;
   1:  PR[GP1:91,2] = PR[GP1:90,2] + -19.847;
   1:L PR[91] 10mm/sec CNT100;
   1:  PR[GP1:91,1] = PR[GP1:90,1] + 9.051;
   1:  PR[GP1:91,2] = PR[GP1:90,2] + -24.581;
   1:L PR[91] 10mm/sec CNT100;
   1:  PR[GP1:91,1] = PR[GP1:90,1] + 11.172;
   1:  PR[GP1:91,2] = PR[GP1:90,2] + -26.150;
   1:L PR[91] 10mm/sec CNT100;
   1:  PR[GP1:91,1] = PR[GP1:90,1] + 15.517;
   1:  PR[GP1:91,2] = PR[GP1:90,2] + -29.541;
   1:L PR[91] 10mm/sec CNT100;
   1:  PR[GP1:91,1] = PR[GP1:90,1] + 18.821;
   1:  PR[GP1:91,2] = PR[GP1:90,2] + -31.338;
   1:L PR[91] 10mm/sec CNT100;
   1:  PR[GP1:91,1] = PR[GP1:90,1] + 25.149;
   1:  PR[GP1:91,2] = PR[GP1:90,2] + -33.567;
   1:L PR[91] 10mm/sec CNT100;
   1:  PR[GP1:91,1] = PR[GP1:90,1] + 27.490;
   1:  PR[GP1:91,2] = PR[GP1:90,2] + -34.328;
   1:L PR[91] 10mm/sec CNT100;
   1:  PR[GP1:91,1] = PR[GP1:90,1] + 29.061;
   1:  PR[GP1:91,2] = PR[GP1:90,2] + -34.558;
   1:L PR[91] 10mm/sec CNT100;
   1:  PR[GP1:91,1] = PR[GP1:90,1] + 38.878;
   1:  PR[GP1:91,2] = PR[GP1:90,2] + -35.048;
   1:L PR[91] 10mm/sec CNT100;
   1:  PR[GP1:91,1] = PR[GP1:90,1] + 49.018;
   1:  PR[GP1:91,2] = PR[GP1:90,2] + -32.767;
   1:L PR[91] 10mm/sec CNT100;
   1:  PR[GP1:91,1] = PR[GP1:90,1] + 51.074;
   1:  PR[GP1:91,2] = PR[GP1:90,2] + -31.735;
   1:L PR[91] 10mm/sec CNT100;
   1:  PR[GP1:91,1] = PR[GP1:90,1] + 58.236;
   1:  PR[GP1:91,2] = PR[GP1:90,2] + -27.705;
   1:L PR[91] 10mm/sec CNT100;
   1:  PR[GP1:91,1] = PR[GP1:90,1] + 61.242;
   1:  PR[GP1:91,2] = PR[GP1:90,2] + -24.751;
   1:L PR[91] 10mm/sec CNT100;
   1:  PR[GP1:91,1] = PR[GP1:90,1] + 65.666;
   1:  PR[GP1:91,2] = PR[GP1:90,2] + -20.077;
   1:L PR[91] 10mm/sec CNT100;
   1:  PR[GP1:91,1] = PR[GP1:90,1] + 68.171;
   1:  PR[GP1:91,2] = PR[GP1:90,2] + -15.280;
   1:L PR[91] 10mm/sec CNT100;
   1:  PR[GP1:91,1] = PR[GP1:90,1] + 70.497;
   1:  PR[GP1:91,2] = PR[GP1:90,2] + -10.597;
   1:L PR[91] 10mm/sec CNT100;
   1:  PR[GP1:91,1] = PR[GP1:90,1] + 71.463;
   1:  PR[GP1:91,2] = PR[GP1:90,2] + -4.633;
   1:L PR[91] 10mm/sec CNT100;
   1:  PR[GP1:91,1] = PR[GP1:90,1] + 71.578;
   1:  PR[GP1:91,2] = PR[GP1:90,2] + -4.044;
   1:L PR[91] 10mm/sec CNT100;
   1:  PR[GP1:91,1] = PR[GP1:90,1] + 72.195;
   1:  PR[GP1:91,2] = PR[GP1:90,2] + -0.008;
   1:L PR[91] 10mm/sec CNT100;
   1:  PR[GP1:91,1] = PR[GP1:90,1] + 71.190;
   1:  PR[GP1:91,2] = PR[GP1:90,2] + 6.029;
   1:L PR[91] 10mm/sec CNT100;
   1:  PR[GP1:91,1] = PR[GP1:90,1] + 70.495;
   1:  PR[GP1:91,2] = PR[GP1:90,2] + 10.590;
   1:L PR[91] 10mm/sec CNT100;
   1:  PR[GP1:91,1] = PR[GP1:90,1] + 68.171;
   1:  PR[GP1:91,2] = PR[GP1:90,2] + 15.271;
   1:L PR[91] 10mm/sec CNT100;
   1:  PR[GP1:91,1] = PR[GP1:90,1] + 65.666;
   1:  PR[GP1:91,2] = PR[GP1:90,2] + 20.068;
   1:L PR[91] 10mm/sec CNT100;
   1:  PR[GP1:91,1] = PR[GP1:90,1] + 61.242;
   1:  PR[GP1:91,2] = PR[GP1:90,2] + 24.742;
   1:L PR[91] 10mm/sec CNT100;
   1:  PR[GP1:91,1] = PR[GP1:90,1] + 58.236;
   1:  PR[GP1:91,2] = PR[GP1:90,2] + 27.696;
   1:L PR[91] 10mm/sec CNT100;
   1:  PR[GP1:91,1] = PR[GP1:90,1] + 51.074;
   1:  PR[GP1:91,2] = PR[GP1:90,2] + 31.726;
   1:L PR[91] 10mm/sec CNT100;
   1:  PR[GP1:91,1] = PR[GP1:90,1] + 49.018;
   1:  PR[GP1:91,2] = PR[GP1:90,2] + 32.758;
   1:L PR[91] 10mm/sec CNT100;
   1:  PR[GP1:91,1] = PR[GP1:90,1] + 38.878;
   1:  PR[GP1:91,2] = PR[GP1:90,2] + 35.039;
   1:L PR[91] 10mm/sec CNT100;
   1:  PR[GP1:91,1] = PR[GP1:90,1] + 29.061;
   1:  PR[GP1:91,2] = PR[GP1:90,2] + 34.549;
   1:L PR[91] 10mm/sec CNT100;
   1:  PR[GP1:91,1] = PR[GP1:90,1] + 27.499;
   1:  PR[GP1:91,2] = PR[GP1:90,2] + 34.321;
   1:L PR[91] 10mm/sec CNT100;
   1:  PR[GP1:91,1] = PR[GP1:90,1] + 21.324;
   1:  PR[GP1:91,2] = PR[GP1:90,2] + 32.114;
   1:L PR[91] 10mm/sec CNT100;
   1:  PR[GP1:91,1] = PR[GP1:90,1] + 18.812;
   1:  PR[GP1:91,2] = PR[GP1:90,2] + 31.324;
   1:L PR[91] 10mm/sec CNT100;
   1:  PR[GP1:91,1] = PR[GP1:90,1] + 15.509;
   1:  PR[GP1:91,2] = PR[GP1:90,2] + 29.528;
   1:L PR[91] 10mm/sec CNT100;
   1:  PR[GP1:91,1] = PR[GP1:90,1] + 12.551;
   1:  PR[GP1:91,2] = PR[GP1:90,2] + 27.359;
   1:L PR[91] 10mm/sec CNT100;
   1:  PR[GP1:91,1] = PR[GP1:90,1] + 9.058;
   1:  PR[GP1:91,2] = PR[GP1:90,2] + 24.580;
   1:L PR[91] 10mm/sec CNT100;
   1:  PR[GP1:91,1] = PR[GP1:90,1] + 5.011;
   1:  PR[GP1:91,2] = PR[GP1:90,2] + 19.838;
   1:L PR[91] 10mm/sec CNT100;
   1:  PR[GP1:91,1] = PR[GP1:90,1] + 4.697;
   1:  PR[GP1:91,2] = PR[GP1:90,2] + 19.407;
   1:L PR[91] 10mm/sec CNT100;
   1:  PR[GP1:91,1] = PR[GP1:90,1] + 4.526;
   1:  PR[GP1:91,2] = PR[GP1:90,2] + 19.220;
   1:L PR[91] 10mm/sec CNT100;
   1:  PR[GP1:91,1] = PR[GP1:90,1] + 0.786;
   1:  PR[GP1:91,2] = PR[GP1:90,2] + 17.037;
   1:L PR[91] 10mm/sec CNT100;
   1:  PR[GP1:91,1] = PR[GP1:90,1] + -3.708;
   1:  PR[GP1:91,2] = PR[GP1:90,2] + 19.981;
   1:  PR[GP1:91,3] = PR[GP1:90,3] + 38.570;
   1:L PR[91] 10mm/sec CNT100;
   1:  PR[GP1:91,1] = PR[GP1:90,1] + -7.768;
   1:  PR[GP1:91,2] = PR[GP1:90,2] + 24.705;
   1:L PR[91] 10mm/sec CNT100;
   1:  PR[GP1:91,1] = PR[GP1:90,1] + -13.583;
   1:  PR[GP1:91,2] = PR[GP1:90,2] + 29.241;
   1:L PR[91] 10mm/sec CNT100;
   1:  PR[GP1:91,1] = PR[GP1:90,1] + -17.971;
   1:  PR[GP1:91,2] = PR[GP1:90,2] + 31.634;
   1:L PR[91] 10mm/sec CNT100;
   1:  PR[GP1:91,1] = PR[GP1:90,1] + -22.284;
   1:  PR[GP1:91,2] = PR[GP1:90,2] + 33.154;
   1:L PR[91] 10mm/sec CNT100;
   1:  PR[GP1:91,1] = PR[GP1:90,1] + -26.013;
   1:  PR[GP1:91,2] = PR[GP1:90,2] + 34.368;
   1:L PR[91] 10mm/sec CNT100;
   1:  PR[GP1:91,1] = PR[GP1:90,1] + -28.548;
   1:  PR[GP1:91,2] = PR[GP1:90,2] + 34.737;
   1:L PR[91] 10mm/sec CNT100;
   1:  PR[GP1:91,1] = PR[GP1:90,1] + -36.570;
   1:  PR[GP1:91,2] = PR[GP1:90,2] + 35.143;
   1:L PR[91] 10mm/sec CNT100;
   1:  PR[GP1:91,1] = PR[GP1:90,1] + -37.772;
   1:  PR[GP1:91,2] = PR[GP1:90,2] + 35.109;
   1:L PR[91] 10mm/sec CNT100;
   1:  PR[GP1:91,1] = PR[GP1:90,1] + -45.240;
   1:  PR[GP1:91,2] = PR[GP1:90,2] + 33.373;
   1:L PR[91] 10mm/sec CNT100;
   1:  PR[GP1:91,1] = PR[GP1:90,1] + -48.182;
   1:  PR[GP1:91,2] = PR[GP1:90,2] + 32.714;
   1:L PR[91] 10mm/sec CNT100;
   1:  PR[GP1:91,1] = PR[GP1:90,1] + -48.777;
   1:  PR[GP1:91,2] = PR[GP1:90,2] + 32.415;
   1:L PR[91] 10mm/sec CNT100;
   1:  PR[GP1:91,1] = PR[GP1:90,1] + -57.308;
   1:  PR[GP1:91,2] = PR[GP1:90,2] + 27.606;
   1:L PR[91] 10mm/sec CNT100;
   1:  PR[GP1:91,1] = PR[GP1:90,1] + -59.239;
   1:  PR[GP1:91,2] = PR[GP1:90,2] + 25.711;
   1:L PR[91] 10mm/sec CNT100;
   1:  PR[GP1:91,1] = PR[GP1:90,1] + -64.661;
   1:  PR[GP1:91,2] = PR[GP1:90,2] + 20.000;
   1:L PR[91] 10mm/sec CNT100;
   1:  PR[GP1:91,1] = PR[GP1:90,1] + -66.521;
   1:  PR[GP1:91,2] = PR[GP1:90,2] + 16.429;
   1:L PR[91] 10mm/sec CNT100;
   1:  PR[GP1:91,1] = PR[GP1:90,1] + -69.440;
   1:  PR[GP1:91,2] = PR[GP1:90,2] + 10.519;
   1:L PR[91] 10mm/sec CNT100;
   1:  PR[GP1:91,1] = PR[GP1:90,1] + -70.196;
   1:  PR[GP1:91,2] = PR[GP1:90,2] + 5.864;
   1:L PR[91] 10mm/sec CNT100;
   1:  PR[GP1:91,1] = PR[GP1:90,1] + -70.286;
   1:  PR[GP1:91,2] = PR[GP1:90,2] + 5.403;
   1:L PR[91] 10mm/sec CNT100;
   1:  PR[GP1:91,1] = PR[GP1:90,1] + -71.114;
   1:  PR[GP1:91,2] = PR[GP1:90,2] + -0.000;
   1:L PR[91] 10mm/sec CNT100;
   1:  PR[GP1:91,1] = PR[GP1:90,1] + -70.311;
   1:  PR[GP1:91,2] = PR[GP1:90,2] + -4.819;
   1:L PR[91] 10mm/sec CNT100;
   1:  PR[GP1:91,1] = PR[GP1:90,1] + -69.439;
   1:  PR[GP1:91,2] = PR[GP1:90,2] + -10.531;
   1:L PR[91] 10mm/sec CNT100;
   1:  PR[GP1:91,1] = PR[GP1:90,1] + -66.521;
   1:  PR[GP1:91,2] = PR[GP1:90,2] + -16.437;
   1:L PR[91] 10mm/sec CNT100;
   1:  PR[GP1:91,1] = PR[GP1:90,1] + -64.661;
   1:  PR[GP1:91,2] = PR[GP1:90,2] + -20.008;
   1:L PR[91] 10mm/sec CNT100;
   1:  PR[GP1:91,1] = PR[GP1:90,1] + -59.239;
   1:  PR[GP1:91,2] = PR[GP1:90,2] + -25.720;
   1:L PR[91] 10mm/sec CNT100;
   1:  PR[GP1:91,1] = PR[GP1:90,1] + -57.308;
   1:  PR[GP1:91,2] = PR[GP1:90,2] + -27.614;
   1:L PR[91] 10mm/sec CNT100;
   1:  PR[GP1:91,1] = PR[GP1:90,1] + -48.777;
   1:  PR[GP1:91,2] = PR[GP1:90,2] + -32.424;
   1:L PR[91] 10mm/sec CNT100;
   1:  PR[GP1:91,1] = PR[GP1:90,1] + -48.182;
   1:  PR[GP1:91,2] = PR[GP1:90,2] + -32.723;
   1:L PR[91] 10mm/sec CNT100;
   1:  PR[GP1:91,1] = PR[GP1:90,1] + -45.239;
   1:  PR[GP1:91,2] = PR[GP1:90,2] + -33.382;
   1:L PR[91] 10mm/sec CNT100;
   1:  PR[GP1:91,1] = PR[GP1:90,1] + -38.589;
   1:  PR[GP1:91,2] = PR[GP1:90,2] + -34.947;
   1:L PR[91] 10mm/sec CNT100;
   1:  PR[GP1:91,1] = PR[GP1:90,1] + -37.778;
   1:  PR[GP1:91,2] = PR[GP1:90,2] + -35.118;
   1:L PR[91] 10mm/sec CNT100;
   1:  PR[GP1:91,1] = PR[GP1:90,1] + -36.570;
   1:  PR[GP1:91,2] = PR[GP1:90,2] + -35.152;
   1:L PR[91] 10mm/sec CNT100;
   1:  PR[GP1:91,1] = PR[GP1:90,1] + -28.548;
   1:  PR[GP1:91,2] = PR[GP1:90,2] + -34.746;
   1:L PR[91] 10mm/sec CNT100;
   1:  PR[GP1:91,1] = PR[GP1:90,1] + -26.022;
   1:  PR[GP1:91,2] = PR[GP1:90,2] + -34.378;
   1:L PR[91] 10mm/sec CNT100;
   1:  PR[GP1:91,1] = PR[GP1:90,1] + -21.262;
   1:  PR[GP1:91,2] = PR[GP1:90,2] + -32.675;
   1:L PR[91] 10mm/sec CNT100;
   1:  PR[GP1:91,1] = PR[GP1:90,1] + -17.962;
   1:  PR[GP1:91,2] = PR[GP1:90,2] + -31.637;
   1:L PR[91] 10mm/sec CNT100;
   1:  PR[GP1:91,1] = PR[GP1:90,1] + -13.575;
   1:  PR[GP1:91,2] = PR[GP1:90,2] + -29.245;
   1:L PR[91] 10mm/sec CNT100;
   1:  PR[GP1:91,1] = PR[GP1:90,1] + -12.093;
   1:  PR[GP1:91,2] = PR[GP1:90,2] + -28.160;
   1:L PR[91] 10mm/sec CNT100;
   1:  PR[GP1:91,1] = PR[GP1:90,1] + -7.770;
   1:  PR[GP1:91,2] = PR[GP1:90,2] + -24.716;
   1:L PR[91] 10mm/sec CNT100;
   1:  PR[GP1:91,1] = PR[GP1:90,1] + -3.653;
   1:  PR[GP1:91,2] = PR[GP1:90,2] + -19.937;
   1:L PR[91] 10mm/sec CNT100;
   1:  PR[GP1:91,1] = PR[GP1:90,1] + -3.310;
   1:  PR[GP1:91,2] = PR[GP1:90,2] + -19.864;
   1:L PR[91] 10mm/sec CNT100;
   1:  PR[GP1:91,1] = PR[GP1:90,1] + 0.414;
   1:  PR[GP1:91,2] = PR[GP1:90,2] + -17.891;
   1:L PR[91] 10mm/sec CNT100;
   1:  PR[GP1:91,1] = PR[GP1:90,1] + 4.541;
   1:  PR[GP1:91,2] = PR[GP1:90,2] + -19.999;
   1:L PR[91] 10mm/sec CNT100;
   1:  PR[GP1:91,1] = PR[GP1:90,1] + 8.640;
   1:  PR[GP1:91,2] = PR[GP1:90,2] + -24.761;
   1:L PR[91] 10mm/sec CNT100;
   1:  PR[GP1:91,1] = PR[GP1:90,1] + 14.423;
   1:  PR[GP1:91,2] = PR[GP1:90,2] + -29.269;
   1:L PR[91] 10mm/sec CNT100;
   1:  PR[GP1:91,1] = PR[GP1:90,1] + 18.782;
   1:  PR[GP1:91,2] = PR[GP1:90,2] + -31.639;
   1:L PR[91] 10mm/sec CNT100;
   1:  PR[GP1:91,1] = PR[GP1:90,1] + 23.094;
   1:  PR[GP1:91,2] = PR[GP1:90,2] + -33.158;
   1:L PR[91] 10mm/sec CNT100;
   1:  PR[GP1:91,1] = PR[GP1:90,1] + 26.832;
   1:  PR[GP1:91,2] = PR[GP1:90,2] + -34.374;
   1:L PR[91] 10mm/sec CNT100;
   1:  PR[GP1:91,1] = PR[GP1:90,1] + 29.364;
   1:  PR[GP1:91,2] = PR[GP1:90,2] + -34.745;
   1:L PR[91] 10mm/sec CNT100;
   1:  PR[GP1:91,1] = PR[GP1:90,1] + 37.388;
   1:  PR[GP1:91,2] = PR[GP1:90,2] + -35.153;
   1:L PR[91] 10mm/sec CNT100;
   1:  PR[GP1:91,1] = PR[GP1:90,1] + 38.586;
   1:  PR[GP1:91,2] = PR[GP1:90,2] + -35.119;
   1:L PR[91] 10mm/sec CNT100;
   1:  PR[GP1:91,1] = PR[GP1:90,1] + 46.061;
   1:  PR[GP1:91,2] = PR[GP1:90,2] + -33.380;
   1:L PR[91] 10mm/sec CNT100;
   1:  PR[GP1:91,1] = PR[GP1:90,1] + 49.002;
   1:  PR[GP1:91,2] = PR[GP1:90,2] + -32.720;
   1:L PR[91] 10mm/sec CNT100;
   1:  PR[GP1:91,1] = PR[GP1:90,1] + 49.597;
   1:  PR[GP1:91,2] = PR[GP1:90,2] + -32.421;
   1:L PR[91] 10mm/sec CNT100;
   1:  PR[GP1:91,1] = PR[GP1:90,1] + 58.127;
   1:  PR[GP1:91,2] = PR[GP1:90,2] + -27.621;
   1:L PR[91] 10mm/sec CNT100;
   1:  PR[GP1:91,1] = PR[GP1:90,1] + 60.058;
   1:  PR[GP1:91,2] = PR[GP1:90,2] + -25.724;
   1:L PR[91] 10mm/sec CNT100;
   1:  PR[GP1:91,1] = PR[GP1:90,1] + 65.481;
   1:  PR[GP1:91,2] = PR[GP1:90,2] + -19.995;
   1:L PR[91] 10mm/sec CNT100;
   1:  PR[GP1:91,1] = PR[GP1:90,1] + 67.341;
   1:  PR[GP1:91,2] = PR[GP1:90,2] + -16.433;
   1:L PR[91] 10mm/sec CNT100;
   1:  PR[GP1:91,1] = PR[GP1:90,1] + 70.261;
   1:  PR[GP1:91,2] = PR[GP1:90,2] + -10.552;
   1:L PR[91] 10mm/sec CNT100;
   1:  PR[GP1:91,1] = PR[GP1:90,1] + 71.016;
   1:  PR[GP1:91,2] = PR[GP1:90,2] + -5.889;
   1:L PR[91] 10mm/sec CNT100;
   1:  PR[GP1:91,1] = PR[GP1:90,1] + 71.106;
   1:  PR[GP1:91,2] = PR[GP1:90,2] + -5.427;
   1:L PR[91] 10mm/sec CNT100;
   1:  PR[GP1:91,1] = PR[GP1:90,1] + 71.935;
   1:  PR[GP1:91,2] = PR[GP1:90,2] + -0.008;
   1:L PR[91] 10mm/sec CNT100;
   1:  PR[GP1:91,1] = PR[GP1:90,1] + 71.131;
   1:  PR[GP1:91,2] = PR[GP1:90,2] + 4.818;
   1:L PR[91] 10mm/sec CNT100;
   1:  PR[GP1:91,1] = PR[GP1:90,1] + 70.259;
   1:  PR[GP1:91,2] = PR[GP1:90,2] + 10.546;
   1:L PR[91] 10mm/sec CNT100;
   1:  PR[GP1:91,1] = PR[GP1:90,1] + 67.341;
   1:  PR[GP1:91,2] = PR[GP1:90,2] + 16.424;
   1:L PR[91] 10mm/sec CNT100;
   1:  PR[GP1:91,1] = PR[GP1:90,1] + 65.481;
   1:  PR[GP1:91,2] = PR[GP1:90,2] + 19.986;
   1:L PR[91] 10mm/sec CNT100;
   1:  PR[GP1:91,1] = PR[GP1:90,1] + 60.058;
   1:  PR[GP1:91,2] = PR[GP1:90,2] + 25.715;
   1:L PR[91] 10mm/sec CNT100;
   1:  PR[GP1:91,1] = PR[GP1:90,1] + 58.127;
   1:  PR[GP1:91,2] = PR[GP1:90,2] + 27.612;
   1:L PR[91] 10mm/sec CNT100;
   1:  PR[GP1:91,1] = PR[GP1:90,1] + 49.597;
   1:  PR[GP1:91,2] = PR[GP1:90,2] + 32.412;
   1:L PR[91] 10mm/sec CNT100;
   1:  PR[GP1:91,1] = PR[GP1:90,1] + 49.002;
   1:  PR[GP1:91,2] = PR[GP1:90,2] + 32.711;
   1:L PR[91] 10mm/sec CNT100;
   1:  PR[GP1:91,1] = PR[GP1:90,1] + 46.060;
   1:  PR[GP1:91,2] = PR[GP1:90,2] + 33.371;
   1:L PR[91] 10mm/sec CNT100;
   1:  PR[GP1:91,1] = PR[GP1:90,1] + 39.405;
   1:  PR[GP1:91,2] = PR[GP1:90,2] + 34.940;
   1:L PR[91] 10mm/sec CNT100;
   1:  PR[GP1:91,1] = PR[GP1:90,1] + 38.593;
   1:  PR[GP1:91,2] = PR[GP1:90,2] + 35.110;
   1:L PR[91] 10mm/sec CNT100;
   1:  PR[GP1:91,1] = PR[GP1:90,1] + 37.388;
   1:  PR[GP1:91,2] = PR[GP1:90,2] + 35.144;
   1:L PR[91] 10mm/sec CNT100;
   1:  PR[GP1:91,1] = PR[GP1:90,1] + 29.365;
   1:  PR[GP1:91,2] = PR[GP1:90,2] + 34.736;
   1:L PR[91] 10mm/sec CNT100;
   1:  PR[GP1:91,1] = PR[GP1:90,1] + 26.841;
   1:  PR[GP1:91,2] = PR[GP1:90,2] + 34.367;
   1:L PR[91] 10mm/sec CNT100;
   1:  PR[GP1:91,1] = PR[GP1:90,1] + 22.081;
   1:  PR[GP1:91,2] = PR[GP1:90,2] + 32.666;
   1:L PR[91] 10mm/sec CNT100;
   1:  PR[GP1:91,1] = PR[GP1:90,1] + 18.773;
   1:  PR[GP1:91,2] = PR[GP1:90,2] + 31.625;
   1:L PR[91] 10mm/sec CNT100;
   1:  PR[GP1:91,1] = PR[GP1:90,1] + 14.415;
   1:  PR[GP1:91,2] = PR[GP1:90,2] + 29.255;
   1:L PR[91] 10mm/sec CNT100;
   1:  PR[GP1:91,1] = PR[GP1:90,1] + 12.929;
   1:  PR[GP1:91,2] = PR[GP1:90,2] + 28.166;
   1:L PR[91] 10mm/sec CNT100;
   1:  PR[GP1:91,1] = PR[GP1:90,1] + 8.642;
   1:  PR[GP1:91,2] = PR[GP1:90,2] + 24.755;
   1:L PR[91] 10mm/sec CNT100;
   1:  PR[GP1:91,1] = PR[GP1:90,1] + 4.541;
   1:  PR[GP1:91,2] = PR[GP1:90,2] + 19.980;
   1:L PR[91] 10mm/sec CNT100;
   1:  PR[GP1:91,1] = PR[GP1:90,1] + 0.419;
   1:  PR[GP1:91,2] = PR[GP1:90,2] + 17.885;
   1:L PR[91] 10mm/sec CNT100;
   1:  PR[GP1:91,1] = PR[GP1:90,1] + 0.039;
   1:  PR[GP1:91,2] = PR[GP1:90,2] + 18.733;
   1:  PR[GP1:91,3] = PR[GP1:90,3] + 39.900;
   1:L PR[91] 10mm/sec CNT100;
   1:  PR[GP1:91,1] = PR[GP1:90,1] + -3.644;
   1:  PR[GP1:91,2] = PR[GP1:90,2] + 20.606;
   1:L PR[91] 10mm/sec CNT100;
   1:  PR[GP1:91,1] = PR[GP1:90,1] + -7.424;
   1:  PR[GP1:91,2] = PR[GP1:90,2] + 25.002;
   1:L PR[91] 10mm/sec CNT100;
   1:  PR[GP1:91,1] = PR[GP1:90,1] + -12.485;
   1:  PR[GP1:91,2] = PR[GP1:90,2] + 28.965;
   1:L PR[91] 10mm/sec CNT100;
   1:  PR[GP1:91,1] = PR[GP1:90,1] + -17.934;
   1:  PR[GP1:91,2] = PR[GP1:90,2] + 31.936;
   1:L PR[91] 10mm/sec CNT100;
   1:  PR[GP1:91,1] = PR[GP1:90,1] + -20.233;
   1:  PR[GP1:91,2] = PR[GP1:90,2] + 32.747;
   1:L PR[91] 10mm/sec CNT100;
   1:  PR[GP1:91,1] = PR[GP1:90,1] + -25.356;
   1:  PR[GP1:91,2] = PR[GP1:90,2] + 34.414;
   1:L PR[91] 10mm/sec CNT100;
   1:  PR[GP1:91,1] = PR[GP1:90,1] + -28.853;
   1:  PR[GP1:91,2] = PR[GP1:90,2] + 34.923;
   1:L PR[91] 10mm/sec CNT100;
   1:  PR[GP1:91,1] = PR[GP1:90,1] + -35.151;
   1:  PR[GP1:91,2] = PR[GP1:90,2] + 35.242;
   1:L PR[91] 10mm/sec CNT100;
   1:  PR[GP1:91,1] = PR[GP1:90,1] + -37.511;
   1:  PR[GP1:91,2] = PR[GP1:90,2] + 35.175;
   1:L PR[91] 10mm/sec CNT100;
   1:  PR[GP1:91,1] = PR[GP1:90,1] + -47.067;
   1:  PR[GP1:91,2] = PR[GP1:90,2] + 32.953;
   1:L PR[91] 10mm/sec CNT100;
   1:  PR[GP1:91,1] = PR[GP1:90,1] + -47.740;
   1:  PR[GP1:91,2] = PR[GP1:90,2] + 32.807;
   1:L PR[91] 10mm/sec CNT100;
   1:  PR[GP1:91,1] = PR[GP1:90,1] + -48.124;
   1:  PR[GP1:91,2] = PR[GP1:90,2] + 32.656;
   1:L PR[91] 10mm/sec CNT100;
   1:  PR[GP1:91,1] = PR[GP1:90,1] + -57.199;
   1:  PR[GP1:91,2] = PR[GP1:90,2] + 27.522;
   1:L PR[91] 10mm/sec CNT100;
   1:  PR[GP1:91,1] = PR[GP1:90,1] + -58.055;
   1:  PR[GP1:91,2] = PR[GP1:90,2] + 26.682;
   1:L PR[91] 10mm/sec CNT100;
   1:  PR[GP1:91,1] = PR[GP1:90,1] + -64.476;
   1:  PR[GP1:91,2] = PR[GP1:90,2] + 19.919;
   1:L PR[91] 10mm/sec CNT100;
   1:  PR[GP1:91,1] = PR[GP1:90,1] + -65.691;
   1:  PR[GP1:91,2] = PR[GP1:90,2] + 17.586;
   1:L PR[91] 10mm/sec CNT100;
   1:  PR[GP1:91,1] = PR[GP1:90,1] + -69.204;
   1:  PR[GP1:91,2] = PR[GP1:90,2] + 10.474;
   1:L PR[91] 10mm/sec CNT100;
   1:  PR[GP1:91,1] = PR[GP1:90,1] + -69.749;
   1:  PR[GP1:91,2] = PR[GP1:90,2] + 7.116;
   1:L PR[91] 10mm/sec CNT100;
   1:  PR[GP1:91,1] = PR[GP1:90,1] + -69.814;
   1:  PR[GP1:91,2] = PR[GP1:90,2] + 6.782;
   1:L PR[91] 10mm/sec CNT100;
   1:  PR[GP1:91,1] = PR[GP1:90,1] + -70.854;
   1:  PR[GP1:91,2] = PR[GP1:90,2] + -0.000;
   1:L PR[91] 10mm/sec CNT100;
   1:  PR[GP1:91,1] = PR[GP1:90,1] + -70.253;
   1:  PR[GP1:91,2] = PR[GP1:90,2] + -3.610;
   1:L PR[91] 10mm/sec CNT100;
   1:  PR[GP1:91,1] = PR[GP1:90,1] + -69.203;
   1:  PR[GP1:91,2] = PR[GP1:90,2] + -10.485;
   1:L PR[91] 10mm/sec CNT100;
   1:  PR[GP1:91,1] = PR[GP1:90,1] + -65.690;
   1:  PR[GP1:91,2] = PR[GP1:90,2] + -17.595;
   1:L PR[91] 10mm/sec CNT100;
   1:  PR[GP1:91,1] = PR[GP1:90,1] + -64.476;
   1:  PR[GP1:91,2] = PR[GP1:90,2] + -19.928;
   1:L PR[91] 10mm/sec CNT100;
   1:  PR[GP1:91,1] = PR[GP1:90,1] + -58.055;
   1:  PR[GP1:91,2] = PR[GP1:90,2] + -26.691;
   1:L PR[91] 10mm/sec CNT100;
   1:  PR[GP1:91,1] = PR[GP1:90,1] + -57.199;
   1:  PR[GP1:91,2] = PR[GP1:90,2] + -27.531;
   1:L PR[91] 10mm/sec CNT100;
   1:  PR[GP1:91,1] = PR[GP1:90,1] + -48.394;
   1:  PR[GP1:91,2] = PR[GP1:90,2] + -32.490;
   1:L PR[91] 10mm/sec CNT100;
   1:  PR[GP1:91,1] = PR[GP1:90,1] + -48.110;
   1:  PR[GP1:91,2] = PR[GP1:90,2] + -32.671;
   1:L PR[91] 10mm/sec CNT100;
   1:  PR[GP1:91,1] = PR[GP1:90,1] + -47.735;
   1:  PR[GP1:91,2] = PR[GP1:90,2] + -32.818;
   1:L PR[91] 10mm/sec CNT100;
   1:  PR[GP1:91,1] = PR[GP1:90,1] + -39.113;
   1:  PR[GP1:91,2] = PR[GP1:90,2] + -34.847;
   1:L PR[91] 10mm/sec CNT100;
   1:  PR[GP1:91,1] = PR[GP1:90,1] + -37.517;
   1:  PR[GP1:91,2] = PR[GP1:90,2] + -35.184;
   1:L PR[91] 10mm/sec CNT100;
   1:  PR[GP1:91,1] = PR[GP1:90,1] + -35.151;
   1:  PR[GP1:91,2] = PR[GP1:90,2] + -35.251;
   1:L PR[91] 10mm/sec CNT100;
   1:  PR[GP1:91,1] = PR[GP1:90,1] + -28.853;
   1:  PR[GP1:91,2] = PR[GP1:90,2] + -34.932;
   1:L PR[91] 10mm/sec CNT100;
   1:  PR[GP1:91,1] = PR[GP1:90,1] + -25.365;
   1:  PR[GP1:91,2] = PR[GP1:90,2] + -34.424;
   1:L PR[91] 10mm/sec CNT100;
   1:  PR[GP1:91,1] = PR[GP1:90,1] + -22.020;
   1:  PR[GP1:91,2] = PR[GP1:90,2] + -33.227;
   1:L PR[91] 10mm/sec CNT100;
   1:  PR[GP1:91,1] = PR[GP1:90,1] + -17.925;
   1:  PR[GP1:91,2] = PR[GP1:90,2] + -31.940;
   1:L PR[91] 10mm/sec CNT100;
   1:  PR[GP1:91,1] = PR[GP1:90,1] + -12.485;
   1:  PR[GP1:91,2] = PR[GP1:90,2] + -28.974;
   1:L PR[91] 10mm/sec CNT100;
   1:  PR[GP1:91,1] = PR[GP1:90,1] + -7.388;
   1:  PR[GP1:91,2] = PR[GP1:90,2] + -24.983;
   1:L PR[91] 10mm/sec CNT100;
   1:  PR[GP1:91,1] = PR[GP1:90,1] + -3.589;
   1:  PR[GP1:91,2] = PR[GP1:90,2] + -20.576;
   1:L PR[91] 10mm/sec CNT100;
   1:  PR[GP1:91,1] = PR[GP1:90,1] + -2.946;
   1:  PR[GP1:91,2] = PR[GP1:90,2] + -20.438;
   1:L PR[91] 10mm/sec CNT100;
   1:  PR[GP1:91,1] = PR[GP1:90,1] + 0.504;
   1:  PR[GP1:91,2] = PR[GP1:90,2] + -18.610;
   1:L PR[91] 10mm/sec CNT100;
   1:  PR[GP1:91,1] = PR[GP1:90,1] + 4.476;
   1:  PR[GP1:91,2] = PR[GP1:90,2] + -20.638;
   1:L PR[91] 10mm/sec CNT100;
   1:  PR[GP1:91,1] = PR[GP1:90,1] + 8.256;
   1:  PR[GP1:91,2] = PR[GP1:90,2] + -25.027;
   1:L PR[91] 10mm/sec CNT100;
   1:  PR[GP1:91,1] = PR[GP1:90,1] + 13.330;
   1:  PR[GP1:91,2] = PR[GP1:90,2] + -28.996;
   1:L PR[91] 10mm/sec CNT100;
   1:  PR[GP1:91,1] = PR[GP1:90,1] + 18.743;
   1:  PR[GP1:91,2] = PR[GP1:90,2] + -31.940;
   1:L PR[91] 10mm/sec CNT100;
   1:  PR[GP1:91,1] = PR[GP1:90,1] + 21.039;
   1:  PR[GP1:91,2] = PR[GP1:90,2] + -32.749;
   1:L PR[91] 10mm/sec CNT100;
   1:  PR[GP1:91,1] = PR[GP1:90,1] + 26.174;
   1:  PR[GP1:91,2] = PR[GP1:90,2] + -34.420;
   1:L PR[91] 10mm/sec CNT100;
   1:  PR[GP1:91,1] = PR[GP1:90,1] + 29.668;
   1:  PR[GP1:91,2] = PR[GP1:90,2] + -34.931;
   1:L PR[91] 10mm/sec CNT100;
   1:  PR[GP1:91,1] = PR[GP1:90,1] + 35.966;
   1:  PR[GP1:91,2] = PR[GP1:90,2] + -35.251;
   1:L PR[91] 10mm/sec CNT100;
   1:  PR[GP1:91,1] = PR[GP1:90,1] + 38.319;
   1:  PR[GP1:91,2] = PR[GP1:90,2] + -35.186;
   1:L PR[91] 10mm/sec CNT100;
   1:  PR[GP1:91,1] = PR[GP1:90,1] + 47.882;
   1:  PR[GP1:91,2] = PR[GP1:90,2] + -32.960;
   1:L PR[91] 10mm/sec CNT100;
   1:  PR[GP1:91,1] = PR[GP1:90,1] + 48.557;
   1:  PR[GP1:91,2] = PR[GP1:90,2] + -32.814;
   1:L PR[91] 10mm/sec CNT100;
   1:  PR[GP1:91,1] = PR[GP1:90,1] + 48.943;
   1:  PR[GP1:91,2] = PR[GP1:90,2] + -32.663;
   1:L PR[91] 10mm/sec CNT100;
   1:  PR[GP1:91,1] = PR[GP1:90,1] + 58.018;
   1:  PR[GP1:91,2] = PR[GP1:90,2] + -27.537;
   1:L PR[91] 10mm/sec CNT100;
   1:  PR[GP1:91,1] = PR[GP1:90,1] + 58.874;
   1:  PR[GP1:91,2] = PR[GP1:90,2] + -26.696;
   1:L PR[91] 10mm/sec CNT100;
   1:  PR[GP1:91,1] = PR[GP1:90,1] + 65.295;
   1:  PR[GP1:91,2] = PR[GP1:90,2] + -19.913;
   1:L PR[91] 10mm/sec CNT100;
   1:  PR[GP1:91,1] = PR[GP1:90,1] + 66.511;
   1:  PR[GP1:91,2] = PR[GP1:90,2] + -17.585;
   1:L PR[91] 10mm/sec CNT100;
   1:  PR[GP1:91,1] = PR[GP1:90,1] + 70.025;
   1:  PR[GP1:91,2] = PR[GP1:90,2] + -10.508;
   1:L PR[91] 10mm/sec CNT100;
   1:  PR[GP1:91,1] = PR[GP1:90,1] + 70.569;
   1:  PR[GP1:91,2] = PR[GP1:90,2] + -7.145;
   1:L PR[91] 10mm/sec CNT100;
   1:  PR[GP1:91,1] = PR[GP1:90,1] + 70.635;
   1:  PR[GP1:91,2] = PR[GP1:90,2] + -6.810;
   1:L PR[91] 10mm/sec CNT100;
   1:  PR[GP1:91,1] = PR[GP1:90,1] + 71.675;
   1:  PR[GP1:91,2] = PR[GP1:90,2] + -0.008;
   1:L PR[91] 10mm/sec CNT100;
   1:  PR[GP1:91,1] = PR[GP1:90,1] + 71.073;
   1:  PR[GP1:91,2] = PR[GP1:90,2] + 3.607;
   1:L PR[91] 10mm/sec CNT100;
   1:  PR[GP1:91,1] = PR[GP1:90,1] + 70.023;
   1:  PR[GP1:91,2] = PR[GP1:90,2] + 10.502;
   1:L PR[91] 10mm/sec CNT100;
   1:  PR[GP1:91,1] = PR[GP1:90,1] + 66.511;
   1:  PR[GP1:91,2] = PR[GP1:90,2] + 17.576;
   1:L PR[91] 10mm/sec CNT100;
   1:  PR[GP1:91,1] = PR[GP1:90,1] + 65.295;
   1:  PR[GP1:91,2] = PR[GP1:90,2] + 19.905;
   1:L PR[91] 10mm/sec CNT100;
   1:  PR[GP1:91,1] = PR[GP1:90,1] + 58.874;
   1:  PR[GP1:91,2] = PR[GP1:90,2] + 26.688;
   1:L PR[91] 10mm/sec CNT100;
   1:  PR[GP1:91,1] = PR[GP1:90,1] + 58.019;
   1:  PR[GP1:91,2] = PR[GP1:90,2] + 27.528;
   1:L PR[91] 10mm/sec CNT100;
   1:  PR[GP1:91,1] = PR[GP1:90,1] + 49.212;
   1:  PR[GP1:91,2] = PR[GP1:90,2] + 32.481;
   1:L PR[91] 10mm/sec CNT100;
   1:  PR[GP1:91,1] = PR[GP1:90,1] + 48.929;
   1:  PR[GP1:91,2] = PR[GP1:90,2] + 32.659;
   1:L PR[91] 10mm/sec CNT100;
   1:  PR[GP1:91,1] = PR[GP1:90,1] + 48.552;
   1:  PR[GP1:91,2] = PR[GP1:90,2] + 32.807;
   1:L PR[91] 10mm/sec CNT100;
   1:  PR[GP1:91,1] = PR[GP1:90,1] + 39.924;
   1:  PR[GP1:91,2] = PR[GP1:90,2] + 34.841;
   1:L PR[91] 10mm/sec CNT100;
   1:  PR[GP1:91,1] = PR[GP1:90,1] + 38.326;
   1:  PR[GP1:91,2] = PR[GP1:90,2] + 35.177;
   1:L PR[91] 10mm/sec CNT100;
   1:  PR[GP1:91,1] = PR[GP1:90,1] + 35.966;
   1:  PR[GP1:91,2] = PR[GP1:90,2] + 35.243;
   1:L PR[91] 10mm/sec CNT100;
   1:  PR[GP1:91,1] = PR[GP1:90,1] + 29.668;
   1:  PR[GP1:91,2] = PR[GP1:90,2] + 34.922;
   1:L PR[91] 10mm/sec CNT100;
   1:  PR[GP1:91,1] = PR[GP1:90,1] + 26.182;
   1:  PR[GP1:91,2] = PR[GP1:90,2] + 34.412;
   1:L PR[91] 10mm/sec CNT100;
   1:  PR[GP1:91,1] = PR[GP1:90,1] + 22.837;
   1:  PR[GP1:91,2] = PR[GP1:90,2] + 33.217;
   1:L PR[91] 10mm/sec CNT100;
   1:  PR[GP1:91,1] = PR[GP1:90,1] + 18.734;
   1:  PR[GP1:91,2] = PR[GP1:90,2] + 31.927;
   1:L PR[91] 10mm/sec CNT100;
   1:  PR[GP1:91,1] = PR[GP1:90,1] + 13.274;
   1:  PR[GP1:91,2] = PR[GP1:90,2] + 28.946;
   1:L PR[91] 10mm/sec CNT100;
   1:  PR[GP1:91,1] = PR[GP1:90,1] + 8.292;
   1:  PR[GP1:91,2] = PR[GP1:90,2] + 25.046;
   1:L PR[91] 10mm/sec CNT100;
   1:  PR[GP1:91,1] = PR[GP1:90,1] + 4.457;
   1:  PR[GP1:91,2] = PR[GP1:90,2] + 20.582;
   1:L PR[91] 10mm/sec CNT100;
   1:  PR[GP1:91,1] = PR[GP1:90,1] + 4.120;
   1:  PR[GP1:91,2] = PR[GP1:90,2] + 20.450;
   1:L PR[91] 10mm/sec CNT100;
   1:  PR[GP1:91,1] = PR[GP1:90,1] + 0.617;
   1:  PR[GP1:91,2] = PR[GP1:90,2] + 18.659;
   1:L PR[91] 10mm/sec CNT100;
   1:  PR[GP1:91,1] = PR[GP1:90,1] + -0.154;
   1:  PR[GP1:91,2] = PR[GP1:90,2] + 19.489;
   1:  PR[GP1:91,3] = PR[GP1:90,3] + 41.230;
   1:L PR[91] 10mm/sec CNT100;
   1:  PR[GP1:91,1] = PR[GP1:90,1] + -3.580;
   1:  PR[GP1:91,2] = PR[GP1:90,2] + 21.231;
   1:L PR[91] 10mm/sec CNT100;
   1:  PR[GP1:91,1] = PR[GP1:90,1] + -7.084;
   1:  PR[GP1:91,2] = PR[GP1:90,2] + 25.306;
   1:L PR[91] 10mm/sec CNT100;
   1:  PR[GP1:91,1] = PR[GP1:90,1] + -11.781;
   1:  PR[GP1:91,2] = PR[GP1:90,2] + 28.984;
   1:L PR[91] 10mm/sec CNT100;
   1:  PR[GP1:91,1] = PR[GP1:90,1] + -11.987;
   1:  PR[GP1:91,2] = PR[GP1:90,2] + 29.129;
   1:L PR[91] 10mm/sec CNT100;
   1:  PR[GP1:91,1] = PR[GP1:90,1] + -17.110;
   1:  PR[GP1:91,2] = PR[GP1:90,2] + 31.810;
   1:L PR[91] 10mm/sec CNT100;
   1:  PR[GP1:91,1] = PR[GP1:90,1] + -17.891;
   1:  PR[GP1:91,2] = PR[GP1:90,2] + 32.236;
   1:L PR[91] 10mm/sec CNT100;
   1:  PR[GP1:91,1] = PR[GP1:90,1] + -24.699;
   1:  PR[GP1:91,2] = PR[GP1:90,2] + 34.460;
   1:L PR[91] 10mm/sec CNT100;
   1:  PR[GP1:91,1] = PR[GP1:90,1] + -29.158;
   1:  PR[GP1:91,2] = PR[GP1:90,2] + 35.109;
   1:L PR[91] 10mm/sec CNT100;
   1:  PR[GP1:91,1] = PR[GP1:90,1] + -33.732;
   1:  PR[GP1:91,2] = PR[GP1:90,2] + 35.341;
   1:L PR[91] 10mm/sec CNT100;
   1:  PR[GP1:91,1] = PR[GP1:90,1] + -37.250;
   1:  PR[GP1:91,2] = PR[GP1:90,2] + 35.241;
   1:L PR[91] 10mm/sec CNT100;
   1:  PR[GP1:91,1] = PR[GP1:90,1] + -44.880;
   1:  PR[GP1:91,2] = PR[GP1:90,2] + 33.467;
   1:L PR[91] 10mm/sec CNT100;
   1:  PR[GP1:91,1] = PR[GP1:90,1] + -46.880;
   1:  PR[GP1:91,2] = PR[GP1:90,2] + 33.034;
   1:L PR[91] 10mm/sec CNT100;
   1:  PR[GP1:91,1] = PR[GP1:90,1] + -48.133;
   1:  PR[GP1:91,2] = PR[GP1:90,2] + 32.541;
   1:L PR[91] 10mm/sec CNT100;
   1:  PR[GP1:91,1] = PR[GP1:90,1] + -56.966;
   1:  PR[GP1:91,2] = PR[GP1:90,2] + 27.514;
   1:L PR[91] 10mm/sec CNT100;
   1:  PR[GP1:91,1] = PR[GP1:90,1] + -57.041;
   1:  PR[GP1:91,2] = PR[GP1:90,2] + 27.468;
   1:L PR[91] 10mm/sec CNT100;
   1:  PR[GP1:91,1] = PR[GP1:90,1] + -57.068;
   1:  PR[GP1:91,2] = PR[GP1:90,2] + 27.443;
   1:L PR[91] 10mm/sec CNT100;
   1:  PR[GP1:91,1] = PR[GP1:90,1] + -64.290;
   1:  PR[GP1:91,2] = PR[GP1:90,2] + 19.839;
   1:L PR[91] 10mm/sec CNT100;
   1:  PR[GP1:91,1] = PR[GP1:90,1] + -64.860;
   1:  PR[GP1:91,2] = PR[GP1:90,2] + 18.743;
   1:L PR[91] 10mm/sec CNT100;
   1:  PR[GP1:91,1] = PR[GP1:90,1] + -68.969;
   1:  PR[GP1:91,2] = PR[GP1:90,2] + 10.427;
   1:L PR[91] 10mm/sec CNT100;
   1:  PR[GP1:91,1] = PR[GP1:90,1] + -69.342;
   1:  PR[GP1:91,2] = PR[GP1:90,2] + 8.170;
   1:L PR[91] 10mm/sec CNT100;
   1:  PR[GP1:91,1] = PR[GP1:90,1] + -70.594;
   1:  PR[GP1:91,2] = PR[GP1:90,2] + -0.000;
   1:L PR[91] 10mm/sec CNT100;
   1:  PR[GP1:91,1] = PR[GP1:90,1] + -70.194;
   1:  PR[GP1:91,2] = PR[GP1:90,2] + -2.401;
   1:L PR[91] 10mm/sec CNT100;
   1:  PR[GP1:91,1] = PR[GP1:90,1] + -68.967;
   1:  PR[GP1:91,2] = PR[GP1:90,2] + -10.440;
   1:L PR[91] 10mm/sec CNT100;
   1:  PR[GP1:91,1] = PR[GP1:90,1] + -64.860;
   1:  PR[GP1:91,2] = PR[GP1:90,2] + -18.752;
   1:L PR[91] 10mm/sec CNT100;
   1:  PR[GP1:91,1] = PR[GP1:90,1] + -64.290;
   1:  PR[GP1:91,2] = PR[GP1:90,2] + -19.847;
   1:L PR[91] 10mm/sec CNT100;
   1:  PR[GP1:91,1] = PR[GP1:90,1] + -57.029;
   1:  PR[GP1:91,2] = PR[GP1:90,2] + -27.480;
   1:L PR[91] 10mm/sec CNT100;
   1:  PR[GP1:91,1] = PR[GP1:90,1] + -48.996;
   1:  PR[GP1:91,2] = PR[GP1:90,2] + -31.999;
   1:L PR[91] 10mm/sec CNT100;
   1:  PR[GP1:91,1] = PR[GP1:90,1] + -48.119;
   1:  PR[GP1:91,2] = PR[GP1:90,2] + -32.555;
   1:L PR[91] 10mm/sec CNT100;
   1:  PR[GP1:91,1] = PR[GP1:90,1] + -46.875;
   1:  PR[GP1:91,2] = PR[GP1:90,2] + -33.044;
   1:L PR[91] 10mm/sec CNT100;
   1:  PR[GP1:91,1] = PR[GP1:90,1] + -39.636;
   1:  PR[GP1:91,2] = PR[GP1:90,2] + -34.748;
   1:L PR[91] 10mm/sec CNT100;
   1:  PR[GP1:91,1] = PR[GP1:90,1] + -37.256;
   1:  PR[GP1:91,2] = PR[GP1:90,2] + -35.250;
   1:L PR[91] 10mm/sec CNT100;
   1:  PR[GP1:91,1] = PR[GP1:90,1] + -33.732;
   1:  PR[GP1:91,2] = PR[GP1:90,2] + -35.350;
   1:L PR[91] 10mm/sec CNT100;
   1:  PR[GP1:91,1] = PR[GP1:90,1] + -29.158;
   1:  PR[GP1:91,2] = PR[GP1:90,2] + -35.118;
   1:L PR[91] 10mm/sec CNT100;
   1:  PR[GP1:91,1] = PR[GP1:90,1] + -24.708;
   1:  PR[GP1:91,2] = PR[GP1:90,2] + -34.471;
   1:L PR[91] 10mm/sec CNT100;
   1:  PR[GP1:91,1] = PR[GP1:90,1] + -22.777;
   1:  PR[GP1:91,2] = PR[GP1:90,2] + -33.780;
   1:L PR[91] 10mm/sec CNT100;
   1:  PR[GP1:91,1] = PR[GP1:90,1] + -17.888;
   1:  PR[GP1:91,2] = PR[GP1:90,2] + -32.243;
   1:L PR[91] 10mm/sec CNT100;
   1:  PR[GP1:91,1] = PR[GP1:90,1] + -17.110;
   1:  PR[GP1:91,2] = PR[GP1:90,2] + -31.819;
   1:L PR[91] 10mm/sec CNT100;
   1:  PR[GP1:91,1] = PR[GP1:90,1] + -11.990;
   1:  PR[GP1:91,2] = PR[GP1:90,2] + -29.140;
   1:L PR[91] 10mm/sec CNT100;
   1:  PR[GP1:91,1] = PR[GP1:90,1] + -11.690;
   1:  PR[GP1:91,2] = PR[GP1:90,2] + -28.922;
   1:L PR[91] 10mm/sec CNT100;
   1:  PR[GP1:91,1] = PR[GP1:90,1] + -7.010;
   1:  PR[GP1:91,2] = PR[GP1:90,2] + -25.257;
   1:L PR[91] 10mm/sec CNT100;
   1:  PR[GP1:91,1] = PR[GP1:90,1] + -3.525;
   1:  PR[GP1:91,2] = PR[GP1:90,2] + -21.215;
   1:L PR[91] 10mm/sec CNT100;
   1:  PR[GP1:91,1] = PR[GP1:90,1] + -2.582;
   1:  PR[GP1:91,2] = PR[GP1:90,2] + -21.012;
   1:L PR[91] 10mm/sec CNT100;
   1:  PR[GP1:91,1] = PR[GP1:90,1] + 0.594;
   1:  PR[GP1:91,2] = PR[GP1:90,2] + -19.329;
   1:L PR[91] 10mm/sec CNT100;
   1:  PR[GP1:91,1] = PR[GP1:90,1] + 4.411;
   1:  PR[GP1:91,2] = PR[GP1:90,2] + -21.277;
   1:L PR[91] 10mm/sec CNT100;
   1:  PR[GP1:91,1] = PR[GP1:90,1] + 7.873;
   1:  PR[GP1:91,2] = PR[GP1:90,2] + -25.298;
   1:L PR[91] 10mm/sec CNT100;
   1:  PR[GP1:91,1] = PR[GP1:90,1] + 12.532;
   1:  PR[GP1:91,2] = PR[GP1:90,2] + -28.943;
   1:L PR[91] 10mm/sec CNT100;
   1:  PR[GP1:91,1] = PR[GP1:90,1] + 12.831;
   1:  PR[GP1:91,2] = PR[GP1:90,2] + -29.159;
   1:L PR[91] 10mm/sec CNT100;
   1:  PR[GP1:91,1] = PR[GP1:90,1] + 17.930;
   1:  PR[GP1:91,2] = PR[GP1:90,2] + -31.821;
   1:L PR[91] 10mm/sec CNT100;
   1:  PR[GP1:91,1] = PR[GP1:90,1] + 18.698;
   1:  PR[GP1:91,2] = PR[GP1:90,2] + -32.238;
   1:L PR[91] 10mm/sec CNT100;
   1:  PR[GP1:91,1] = PR[GP1:90,1] + 25.516;
   1:  PR[GP1:91,2] = PR[GP1:90,2] + -34.466;
   1:L PR[91] 10mm/sec CNT100;
   1:  PR[GP1:91,1] = PR[GP1:90,1] + 29.971;
   1:  PR[GP1:91,2] = PR[GP1:90,2] + -35.118;
   1:L PR[91] 10mm/sec CNT100;
   1:  PR[GP1:91,1] = PR[GP1:90,1] + 34.544;
   1:  PR[GP1:91,2] = PR[GP1:90,2] + -35.350;
   1:L PR[91] 10mm/sec CNT100;
   1:  PR[GP1:91,1] = PR[GP1:90,1] + 38.052;
   1:  PR[GP1:91,2] = PR[GP1:90,2] + -35.253;
   1:L PR[91] 10mm/sec CNT100;
   1:  PR[GP1:91,1] = PR[GP1:90,1] + 45.684;
   1:  PR[GP1:91,2] = PR[GP1:90,2] + -33.476;
   1:L PR[91] 10mm/sec CNT100;
   1:  PR[GP1:91,1] = PR[GP1:90,1] + 47.689;
   1:  PR[GP1:91,2] = PR[GP1:90,2] + -33.043;
   1:L PR[91] 10mm/sec CNT100;
   1:  PR[GP1:91,1] = PR[GP1:90,1] + 48.947;
   1:  PR[GP1:91,2] = PR[GP1:90,2] + -32.550;
   1:L PR[91] 10mm/sec CNT100;
   1:  PR[GP1:91,1] = PR[GP1:90,1] + 57.786;
   1:  PR[GP1:91,2] = PR[GP1:90,2] + -27.529;
   1:L PR[91] 10mm/sec CNT100;
   1:  PR[GP1:91,1] = PR[GP1:90,1] + 57.861;
   1:  PR[GP1:91,2] = PR[GP1:90,2] + -27.483;
   1:L PR[91] 10mm/sec CNT100;
   1:  PR[GP1:91,1] = PR[GP1:90,1] + 57.887;
   1:  PR[GP1:91,2] = PR[GP1:90,2] + -27.459;
   1:L PR[91] 10mm/sec CNT100;
   1:  PR[GP1:91,1] = PR[GP1:90,1] + 65.110;
   1:  PR[GP1:91,2] = PR[GP1:90,2] + -19.831;
   1:L PR[91] 10mm/sec CNT100;
   1:  PR[GP1:91,1] = PR[GP1:90,1] + 65.681;
   1:  PR[GP1:91,2] = PR[GP1:90,2] + -18.738;
   1:L PR[91] 10mm/sec CNT100;
   1:  PR[GP1:91,1] = PR[GP1:90,1] + 69.789;
   1:  PR[GP1:91,2] = PR[GP1:90,2] + -10.463;
   1:L PR[91] 10mm/sec CNT100;
   1:  PR[GP1:91,1] = PR[GP1:90,1] + 70.162;
   1:  PR[GP1:91,2] = PR[GP1:90,2] + -8.202;
   1:L PR[91] 10mm/sec CNT100;
   1:  PR[GP1:91,1] = PR[GP1:90,1] + 71.415;
   1:  PR[GP1:91,2] = PR[GP1:90,2] + -0.008;
   1:L PR[91] 10mm/sec CNT100;
   1:  PR[GP1:91,1] = PR[GP1:90,1] + 71.015;
   1:  PR[GP1:91,2] = PR[GP1:90,2] + 2.396;
   1:L PR[91] 10mm/sec CNT100;
   1:  PR[GP1:91,1] = PR[GP1:90,1] + 69.787;
   1:  PR[GP1:91,2] = PR[GP1:90,2] + 10.457;
   1:L PR[91] 10mm/sec CNT100;
   1:  PR[GP1:91,1] = PR[GP1:90,1] + 65.681;
   1:  PR[GP1:91,2] = PR[GP1:90,2] + 18.729;
   1:L PR[91] 10mm/sec CNT100;
   1:  PR[GP1:91,1] = PR[GP1:90,1] + 65.110;
   1:  PR[GP1:91,2] = PR[GP1:90,2] + 19.822;
   1:L PR[91] 10mm/sec CNT100;
   1:  PR[GP1:91,1] = PR[GP1:90,1] + 57.848;
   1:  PR[GP1:91,2] = PR[GP1:90,2] + 27.478;
   1:L PR[91] 10mm/sec CNT100;
   1:  PR[GP1:91,1] = PR[GP1:90,1] + 49.808;
   1:  PR[GP1:91,2] = PR[GP1:90,2] + 31.996;
   1:L PR[91] 10mm/sec CNT100;
   1:  PR[GP1:91,1] = PR[GP1:90,1] + 48.935;
   1:  PR[GP1:91,2] = PR[GP1:90,2] + 32.546;
   1:L PR[91] 10mm/sec CNT100;
   1:  PR[GP1:91,1] = PR[GP1:90,1] + 47.684;
   1:  PR[GP1:91,2] = PR[GP1:90,2] + 33.036;
   1:L PR[91] 10mm/sec CNT100;
   1:  PR[GP1:91,1] = PR[GP1:90,1] + 40.442;
   1:  PR[GP1:91,2] = PR[GP1:90,2] + 34.743;
   1:L PR[91] 10mm/sec CNT100;
   1:  PR[GP1:91,1] = PR[GP1:90,1] + 38.059;
   1:  PR[GP1:91,2] = PR[GP1:90,2] + 35.244;
   1:L PR[91] 10mm/sec CNT100;
   1:  PR[GP1:91,1] = PR[GP1:90,1] + 34.544;
   1:  PR[GP1:91,2] = PR[GP1:90,2] + 35.341;
   1:L PR[91] 10mm/sec CNT100;
   1:  PR[GP1:91,1] = PR[GP1:90,1] + 29.971;
   1:  PR[GP1:91,2] = PR[GP1:90,2] + 35.109;
   1:L PR[91] 10mm/sec CNT100;
   1:  PR[GP1:91,1] = PR[GP1:90,1] + 25.524;
   1:  PR[GP1:91,2] = PR[GP1:90,2] + 34.458;
   1:L PR[91] 10mm/sec CNT100;
   1:  PR[GP1:91,1] = PR[GP1:90,1] + 23.594;
   1:  PR[GP1:91,2] = PR[GP1:90,2] + 33.768;
   1:L PR[91] 10mm/sec CNT100;
   1:  PR[GP1:91,1] = PR[GP1:90,1] + 18.695;
   1:  PR[GP1:91,2] = PR[GP1:90,2] + 32.228;
   1:L PR[91] 10mm/sec CNT100;
   1:  PR[GP1:91,1] = PR[GP1:90,1] + 17.930;
   1:  PR[GP1:91,2] = PR[GP1:90,2] + 31.812;
   1:L PR[91] 10mm/sec CNT100;
   1:  PR[GP1:91,1] = PR[GP1:90,1] + 12.827;
   1:  PR[GP1:91,2] = PR[GP1:90,2] + 29.149;
   1:L PR[91] 10mm/sec CNT100;
   1:  PR[GP1:91,1] = PR[GP1:90,1] + 12.622;
   1:  PR[GP1:91,2] = PR[GP1:90,2] + 29.004;
   1:L PR[91] 10mm/sec CNT100;
   1:  PR[GP1:91,1] = PR[GP1:90,1] + 7.948;
   1:  PR[GP1:91,2] = PR[GP1:90,2] + 25.347;
   1:L PR[91] 10mm/sec CNT100;
   1:  PR[GP1:91,1] = PR[GP1:90,1] + 4.392;
   1:  PR[GP1:91,2] = PR[GP1:90,2] + 21.208;
   1:L PR[91] 10mm/sec CNT100;
   1:  PR[GP1:91,1] = PR[GP1:90,1] + 3.927;
   1:  PR[GP1:91,2] = PR[GP1:90,2] + 21.024;
   1:L PR[91] 10mm/sec CNT100;
   1:  PR[GP1:91,1] = PR[GP1:90,1] + 0.706;
   1:  PR[GP1:91,2] = PR[GP1:90,2] + 19.378;
   1:L PR[91] 10mm/sec CNT100;
   1:  PR[GP1:91,1] = PR[GP1:90,1] + -0.347;
   1:  PR[GP1:91,2] = PR[GP1:90,2] + 20.244;
   1:  PR[GP1:91,3] = PR[GP1:90,3] + 42.560;
   1:L PR[91] 10mm/sec CNT100;
   1:  PR[GP1:91,1] = PR[GP1:90,1] + -3.516;
   1:  PR[GP1:91,2] = PR[GP1:90,2] + 21.856;
   1:L PR[91] 10mm/sec CNT100;
   1:  PR[GP1:91,1] = PR[GP1:90,1] + -6.745;
   1:  PR[GP1:91,2] = PR[GP1:90,2] + 25.610;
   1:L PR[91] 10mm/sec CNT100;
   1:  PR[GP1:91,1] = PR[GP1:90,1] + -11.062;
   1:  PR[GP1:91,2] = PR[GP1:90,2] + 28.991;
   1:L PR[91] 10mm/sec CNT100;
   1:  PR[GP1:91,1] = PR[GP1:90,1] + -11.527;
   1:  PR[GP1:91,2] = PR[GP1:90,2] + 29.320;
   1:L PR[91] 10mm/sec CNT100;
   1:  PR[GP1:91,1] = PR[GP1:90,1] + -17.258;
   1:  PR[GP1:91,2] = PR[GP1:90,2] + 32.318;
   1:L PR[91] 10mm/sec CNT100;
   1:  PR[GP1:91,1] = PR[GP1:90,1] + -24.041;
   1:  PR[GP1:91,2] = PR[GP1:90,2] + 34.507;
   1:L PR[91] 10mm/sec CNT100;
   1:  PR[GP1:91,1] = PR[GP1:90,1] + -29.463;
   1:  PR[GP1:91,2] = PR[GP1:90,2] + 35.295;
   1:L PR[91] 10mm/sec CNT100;
   1:  PR[GP1:91,1] = PR[GP1:90,1] + -32.313;
   1:  PR[GP1:91,2] = PR[GP1:90,2] + 35.440;
   1:L PR[91] 10mm/sec CNT100;
   1:  PR[GP1:91,1] = PR[GP1:90,1] + -36.989;
   1:  PR[GP1:91,2] = PR[GP1:90,2] + 35.307;
   1:L PR[91] 10mm/sec CNT100;
   1:  PR[GP1:91,1] = PR[GP1:90,1] + -42.693;
   1:  PR[GP1:91,2] = PR[GP1:90,2] + 33.981;
   1:L PR[91] 10mm/sec CNT100;
   1:  PR[GP1:91,1] = PR[GP1:90,1] + -46.020;
   1:  PR[GP1:91,2] = PR[GP1:90,2] + 33.260;
   1:L PR[91] 10mm/sec CNT100;
   1:  PR[GP1:91,1] = PR[GP1:90,1] + -48.142;
   1:  PR[GP1:91,2] = PR[GP1:90,2] + 32.425;
   1:L PR[91] 10mm/sec CNT100;
   1:  PR[GP1:91,1] = PR[GP1:90,1] + -55.606;
   1:  PR[GP1:91,2] = PR[GP1:90,2] + 28.178;
   1:L PR[91] 10mm/sec CNT100;
   1:  PR[GP1:91,1] = PR[GP1:90,1] + -56.576;
   1:  PR[GP1:91,2] = PR[GP1:90,2] + 27.577;
   1:L PR[91] 10mm/sec CNT100;
   1:  PR[GP1:91,1] = PR[GP1:90,1] + -57.190;
   1:  PR[GP1:91,2] = PR[GP1:90,2] + 27.026;
   1:L PR[91] 10mm/sec CNT100;
   1:  PR[GP1:91,1] = PR[GP1:90,1] + -64.095;
   1:  PR[GP1:91,2] = PR[GP1:90,2] + 19.760;
   1:L PR[91] 10mm/sec CNT100;
   1:  PR[GP1:91,1] = PR[GP1:90,1] + -68.731;
   1:  PR[GP1:91,2] = PR[GP1:90,2] + 10.385;
   1:L PR[91] 10mm/sec CNT100;
   1:  PR[GP1:91,1] = PR[GP1:90,1] + -70.334;
   1:  PR[GP1:91,2] = PR[GP1:90,2] + -0.001;
   1:L PR[91] 10mm/sec CNT100;
   1:  PR[GP1:91,1] = PR[GP1:90,1] + -70.136;
   1:  PR[GP1:91,2] = PR[GP1:90,2] + -1.191;
   1:L PR[91] 10mm/sec CNT100;
   1:  PR[GP1:91,1] = PR[GP1:90,1] + -68.731;
   1:  PR[GP1:91,2] = PR[GP1:90,2] + -10.394;
   1:L PR[91] 10mm/sec CNT100;
   1:  PR[GP1:91,1] = PR[GP1:90,1] + -64.095;
   1:  PR[GP1:91,2] = PR[GP1:90,2] + -19.769;
   1:L PR[91] 10mm/sec CNT100;
   1:  PR[GP1:91,1] = PR[GP1:90,1] + -57.190;
   1:  PR[GP1:91,2] = PR[GP1:90,2] + -27.035;
   1:L PR[91] 10mm/sec CNT100;
   1:  PR[GP1:91,1] = PR[GP1:90,1] + -56.586;
   1:  PR[GP1:91,2] = PR[GP1:90,2] + -27.577;
   1:L PR[91] 10mm/sec CNT100;
   1:  PR[GP1:91,1] = PR[GP1:90,1] + -49.597;
   1:  PR[GP1:91,2] = PR[GP1:90,2] + -31.508;
   1:L PR[91] 10mm/sec CNT100;
   1:  PR[GP1:91,1] = PR[GP1:90,1] + -48.128;
   1:  PR[GP1:91,2] = PR[GP1:90,2] + -32.439;
   1:L PR[91] 10mm/sec CNT100;
   1:  PR[GP1:91,1] = PR[GP1:90,1] + -46.015;
   1:  PR[GP1:91,2] = PR[GP1:90,2] + -33.270;
   1:L PR[91] 10mm/sec CNT100;
   1:  PR[GP1:91,1] = PR[GP1:90,1] + -40.160;
   1:  PR[GP1:91,2] = PR[GP1:90,2] + -34.649;
   1:L PR[91] 10mm/sec CNT100;
   1:  PR[GP1:91,1] = PR[GP1:90,1] + -36.995;
   1:  PR[GP1:91,2] = PR[GP1:90,2] + -35.316;
   1:L PR[91] 10mm/sec CNT100;
   1:  PR[GP1:91,1] = PR[GP1:90,1] + -32.313;
   1:  PR[GP1:91,2] = PR[GP1:90,2] + -35.449;
   1:L PR[91] 10mm/sec CNT100;
   1:  PR[GP1:91,1] = PR[GP1:90,1] + -29.463;
   1:  PR[GP1:91,2] = PR[GP1:90,2] + -35.304;
   1:L PR[91] 10mm/sec CNT100;
   1:  PR[GP1:91,1] = PR[GP1:90,1] + -24.050;
   1:  PR[GP1:91,2] = PR[GP1:90,2] + -34.517;
   1:L PR[91] 10mm/sec CNT100;
   1:  PR[GP1:91,1] = PR[GP1:90,1] + -23.534;
   1:  PR[GP1:91,2] = PR[GP1:90,2] + -34.332;
   1:L PR[91] 10mm/sec CNT100;
   1:  PR[GP1:91,1] = PR[GP1:90,1] + -17.711;
   1:  PR[GP1:91,2] = PR[GP1:90,2] + -32.485;
   1:L PR[91] 10mm/sec CNT100;
   1:  PR[GP1:91,1] = PR[GP1:90,1] + -17.263;
   1:  PR[GP1:91,2] = PR[GP1:90,2] + -32.330;
   1:L PR[91] 10mm/sec CNT100;
   1:  PR[GP1:91,1] = PR[GP1:90,1] + -11.530;
   1:  PR[GP1:91,2] = PR[GP1:90,2] + -29.330;
   1:L PR[91] 10mm/sec CNT100;
   1:  PR[GP1:91,1] = PR[GP1:90,1] + -10.874;
   1:  PR[GP1:91,2] = PR[GP1:90,2] + -28.854;
   1:L PR[91] 10mm/sec CNT100;
   1:  PR[GP1:91,1] = PR[GP1:90,1] + -6.632;
   1:  PR[GP1:91,2] = PR[GP1:90,2] + -25.532;
   1:L PR[91] 10mm/sec CNT100;
   1:  PR[GP1:91,1] = PR[GP1:90,1] + -3.461;
   1:  PR[GP1:91,2] = PR[GP1:90,2] + -21.853;
   1:L PR[91] 10mm/sec CNT100;
   1:  PR[GP1:91,1] = PR[GP1:90,1] + -2.218;
   1:  PR[GP1:91,2] = PR[GP1:90,2] + -21.587;
   1:L PR[91] 10mm/sec CNT100;
   1:  PR[GP1:91,1] = PR[GP1:90,1] + 0.683;
   1:  PR[GP1:91,2] = PR[GP1:90,2] + -20.049;
   1:L PR[91] 10mm/sec CNT100;
   1:  PR[GP1:91,1] = PR[GP1:90,1] + 4.345;
   1:  PR[GP1:91,2] = PR[GP1:90,2] + -21.916;
   1:L PR[91] 10mm/sec CNT100;
   1:  PR[GP1:91,1] = PR[GP1:90,1] + 7.491;
   1:  PR[GP1:91,2] = PR[GP1:90,2] + -25.569;
   1:L PR[91] 10mm/sec CNT100;
   1:  PR[GP1:91,1] = PR[GP1:90,1] + 11.713;
   1:  PR[GP1:91,2] = PR[GP1:90,2] + -28.872;
   1:L PR[91] 10mm/sec CNT100;
   1:  PR[GP1:91,1] = PR[GP1:90,1] + 12.369;
   1:  PR[GP1:91,2] = PR[GP1:90,2] + -29.349;
   1:L PR[91] 10mm/sec CNT100;
   1:  PR[GP1:91,1] = PR[GP1:90,1] + 18.062;
   1:  PR[GP1:91,2] = PR[GP1:90,2] + -32.320;
   1:L PR[91] 10mm/sec CNT100;
   1:  PR[GP1:91,1] = PR[GP1:90,1] + 24.856;
   1:  PR[GP1:91,2] = PR[GP1:90,2] + -34.511;
   1:L PR[91] 10mm/sec CNT100;
   1:  PR[GP1:91,1] = PR[GP1:90,1] + 30.274;
   1:  PR[GP1:91,2] = PR[GP1:90,2] + -35.304;
   1:L PR[91] 10mm/sec CNT100;
   1:  PR[GP1:91,1] = PR[GP1:90,1] + 33.122;
   1:  PR[GP1:91,2] = PR[GP1:90,2] + -35.449;
   1:L PR[91] 10mm/sec CNT100;
   1:  PR[GP1:91,1] = PR[GP1:90,1] + 37.785;
   1:  PR[GP1:91,2] = PR[GP1:90,2] + -35.319;
   1:L PR[91] 10mm/sec CNT100;
   1:  PR[GP1:91,1] = PR[GP1:90,1] + 43.487;
   1:  PR[GP1:91,2] = PR[GP1:90,2] + -33.992;
   1:L PR[91] 10mm/sec CNT100;
   1:  PR[GP1:91,1] = PR[GP1:90,1] + 46.822;
   1:  PR[GP1:91,2] = PR[GP1:90,2] + -33.271;
   1:L PR[91] 10mm/sec CNT100;
   1:  PR[GP1:91,1] = PR[GP1:90,1] + 48.952;
   1:  PR[GP1:91,2] = PR[GP1:90,2] + -32.437;
   1:L PR[91] 10mm/sec CNT100;
   1:  PR[GP1:91,1] = PR[GP1:90,1] + 56.419;
   1:  PR[GP1:91,2] = PR[GP1:90,2] + -28.195;
   1:L PR[91] 10mm/sec CNT100;
   1:  PR[GP1:91,1] = PR[GP1:90,1] + 57.387;
   1:  PR[GP1:91,2] = PR[GP1:90,2] + -27.598;
   1:L PR[91] 10mm/sec CNT100;
   1:  PR[GP1:91,1] = PR[GP1:90,1] + 58.000;
   1:  PR[GP1:91,2] = PR[GP1:90,2] + -27.051;
   1:L PR[91] 10mm/sec CNT100;
   1:  PR[GP1:91,1] = PR[GP1:90,1] + 64.892;
   1:  PR[GP1:91,2] = PR[GP1:90,2] + -19.783;
   1:L PR[91] 10mm/sec CNT100;
   1:  PR[GP1:91,1] = PR[GP1:90,1] + 65.215;
   1:  PR[GP1:91,2] = PR[GP1:90,2] + -19.156;
   1:L PR[91] 10mm/sec CNT100;
   1:  PR[GP1:91,1] = PR[GP1:90,1] + 69.553;
   1:  PR[GP1:91,2] = PR[GP1:90,2] + -10.418;
   1:L PR[91] 10mm/sec CNT100;
   1:  PR[GP1:91,1] = PR[GP1:90,1] + 69.691;
   1:  PR[GP1:91,2] = PR[GP1:90,2] + -9.586;
   1:L PR[91] 10mm/sec CNT100;
   1:  PR[GP1:91,1] = PR[GP1:90,1] + 71.155;
   1:  PR[GP1:91,2] = PR[GP1:90,2] + -0.008;
   1:L PR[91] 10mm/sec CNT100;
   1:  PR[GP1:91,1] = PR[GP1:90,1] + 70.956;
   1:  PR[GP1:91,2] = PR[GP1:90,2] + 1.185;
   1:L PR[91] 10mm/sec CNT100;
   1:  PR[GP1:91,1] = PR[GP1:90,1] + 69.551;
   1:  PR[GP1:91,2] = PR[GP1:90,2] + 10.413;
   1:L PR[91] 10mm/sec CNT100;
   1:  PR[GP1:91,1] = PR[GP1:90,1] + 64.915;
   1:  PR[GP1:91,2] = PR[GP1:90,2] + 19.743;
   1:L PR[91] 10mm/sec CNT100;
   1:  PR[GP1:91,1] = PR[GP1:90,1] + 58.000;
   1:  PR[GP1:91,2] = PR[GP1:90,2] + 27.042;
   1:L PR[91] 10mm/sec CNT100;
   1:  PR[GP1:91,1] = PR[GP1:90,1] + 57.397;
   1:  PR[GP1:91,2] = PR[GP1:90,2] + 27.581;
   1:L PR[91] 10mm/sec CNT100;
   1:  PR[GP1:91,1] = PR[GP1:90,1] + 50.404;
   1:  PR[GP1:91,2] = PR[GP1:90,2] + 31.510;
   1:L PR[91] 10mm/sec CNT100;
   1:  PR[GP1:91,1] = PR[GP1:90,1] + 48.940;
   1:  PR[GP1:91,2] = PR[GP1:90,2] + 32.433;
   1:L PR[91] 10mm/sec CNT100;
   1:  PR[GP1:91,1] = PR[GP1:90,1] + 46.816;
   1:  PR[GP1:91,2] = PR[GP1:90,2] + 33.264;
   1:L PR[91] 10mm/sec CNT100;
   1:  PR[GP1:91,1] = PR[GP1:90,1] + 40.961;
   1:  PR[GP1:91,2] = PR[GP1:90,2] + 34.644;
   1:L PR[91] 10mm/sec CNT100;
   1:  PR[GP1:91,1] = PR[GP1:90,1] + 37.792;
   1:  PR[GP1:91,2] = PR[GP1:90,2] + 35.310;
   1:L PR[91] 10mm/sec CNT100;
   1:  PR[GP1:91,1] = PR[GP1:90,1] + 33.122;
   1:  PR[GP1:91,2] = PR[GP1:90,2] + 35.440;
   1:L PR[91] 10mm/sec CNT100;
   1:  PR[GP1:91,1] = PR[GP1:90,1] + 30.274;
   1:  PR[GP1:91,2] = PR[GP1:90,2] + 35.295;
   1:L PR[91] 10mm/sec CNT100;
   1:  PR[GP1:91,1] = PR[GP1:90,1] + 24.866;
   1:  PR[GP1:91,2] = PR[GP1:90,2] + 34.504;
   1:L PR[91] 10mm/sec CNT100;
   1:  PR[GP1:91,1] = PR[GP1:90,1] + 24.351;
   1:  PR[GP1:91,2] = PR[GP1:90,2] + 34.320;
   1:L PR[91] 10mm/sec CNT100;
   1:  PR[GP1:91,1] = PR[GP1:90,1] + 18.518;
   1:  PR[GP1:91,2] = PR[GP1:90,2] + 32.470;
   1:L PR[91] 10mm/sec CNT100;
   1:  PR[GP1:91,1] = PR[GP1:90,1] + 18.069;
   1:  PR[GP1:91,2] = PR[GP1:90,2] + 32.314;
   1:L PR[91] 10mm/sec CNT100;
   1:  PR[GP1:91,1] = PR[GP1:90,1] + 12.367;
   1:  PR[GP1:91,2] = PR[GP1:90,2] + 29.339;
   1:L PR[91] 10mm/sec CNT100;
   1:  PR[GP1:91,1] = PR[GP1:90,1] + 11.902;
   1:  PR[GP1:91,2] = PR[GP1:90,2] + 29.010;
   1:L PR[91] 10mm/sec CNT100;
   1:  PR[GP1:91,1] = PR[GP1:90,1] + 7.604;
   1:  PR[GP1:91,2] = PR[GP1:90,2] + 25.647;
   1:L PR[91] 10mm/sec CNT100;
   1:  PR[GP1:91,1] = PR[GP1:90,1] + 4.327;
   1:  PR[GP1:91,2] = PR[GP1:90,2] + 21.833;
   1:L PR[91] 10mm/sec CNT100;
   1:  PR[GP1:91,1] = PR[GP1:90,1] + 3.733;
   1:  PR[GP1:91,2] = PR[GP1:90,2] + 21.598;
   1:L PR[91] 10mm/sec CNT100;
   1:  PR[GP1:91,1] = PR[GP1:90,1] + 0.796;
   1:  PR[GP1:91,2] = PR[GP1:90,2] + 20.097;
   1:L PR[91] 10mm/sec CNT100;
   1:  PR[GP1:91,1] = PR[GP1:90,1] + -0.541;
   1:  PR[GP1:91,2] = PR[GP1:90,2] + 21.000;
   1:  PR[GP1:91,3] = PR[GP1:90,3] + 43.890;
   1:L PR[91] 10mm/sec CNT100;
   1:  PR[GP1:91,1] = PR[GP1:90,1] + -3.453;
   1:  PR[GP1:91,2] = PR[GP1:90,2] + 22.481;
   1:L PR[91] 10mm/sec CNT100;
   1:  PR[GP1:91,1] = PR[GP1:90,1] + -6.405;
   1:  PR[GP1:91,2] = PR[GP1:90,2] + 25.914;
   1:L PR[91] 10mm/sec CNT100;
   1:  PR[GP1:91,1] = PR[GP1:90,1] + -10.344;
   1:  PR[GP1:91,2] = PR[GP1:90,2] + 28.999;
   1:L PR[91] 10mm/sec CNT100;
   1:  PR[GP1:91,1] = PR[GP1:90,1] + -11.068;
   1:  PR[GP1:91,2] = PR[GP1:90,2] + 29.510;
   1:L PR[91] 10mm/sec CNT100;
   1:  PR[GP1:91,1] = PR[GP1:90,1] + -16.513;
   1:  PR[GP1:91,2] = PR[GP1:90,2] + 32.359;
   1:L PR[91] 10mm/sec CNT100;
   1:  PR[GP1:91,1] = PR[GP1:90,1] + -23.515;
   1:  PR[GP1:91,2] = PR[GP1:90,2] + 34.618;
   1:L PR[91] 10mm/sec CNT100;
   1:  PR[GP1:91,1] = PR[GP1:90,1] + -26.665;
   1:  PR[GP1:91,2] = PR[GP1:90,2] + 35.030;
   1:L PR[91] 10mm/sec CNT100;
   1:  PR[GP1:91,1] = PR[GP1:90,1] + -29.768;
   1:  PR[GP1:91,2] = PR[GP1:90,2] + 35.481;
   1:L PR[91] 10mm/sec CNT100;
   1:  PR[GP1:91,1] = PR[GP1:90,1] + -30.894;
   1:  PR[GP1:91,2] = PR[GP1:90,2] + 35.539;
   1:L PR[91] 10mm/sec CNT100;
   1:  PR[GP1:91,1] = PR[GP1:90,1] + -36.728;
   1:  PR[GP1:91,2] = PR[GP1:90,2] + 35.373;
   1:L PR[91] 10mm/sec CNT100;
   1:  PR[GP1:91,1] = PR[GP1:90,1] + -40.506;
   1:  PR[GP1:91,2] = PR[GP1:90,2] + 34.494;
   1:L PR[91] 10mm/sec CNT100;
   1:  PR[GP1:91,1] = PR[GP1:90,1] + -45.160;
   1:  PR[GP1:91,2] = PR[GP1:90,2] + 33.486;
   1:L PR[91] 10mm/sec CNT100;
   1:  PR[GP1:91,1] = PR[GP1:90,1] + -48.151;
   1:  PR[GP1:91,2] = PR[GP1:90,2] + 32.309;
   1:L PR[91] 10mm/sec CNT100;
   1:  PR[GP1:91,1] = PR[GP1:90,1] + -54.245;
   1:  PR[GP1:91,2] = PR[GP1:90,2] + 28.841;
   1:L PR[91] 10mm/sec CNT100;
   1:  PR[GP1:91,1] = PR[GP1:90,1] + -56.111;
   1:  PR[GP1:91,2] = PR[GP1:90,2] + 27.685;
   1:L PR[91] 10mm/sec CNT100;
   1:  PR[GP1:91,1] = PR[GP1:90,1] + -57.312;
   1:  PR[GP1:91,2] = PR[GP1:90,2] + 26.609;
   1:L PR[91] 10mm/sec CNT100;
   1:  PR[GP1:91,1] = PR[GP1:90,1] + -63.310;
   1:  PR[GP1:91,2] = PR[GP1:90,2] + 20.303;
   1:L PR[91] 10mm/sec CNT100;
   1:  PR[GP1:91,1] = PR[GP1:90,1] + -63.810;
   1:  PR[GP1:91,2] = PR[GP1:90,2] + 19.654;
   1:L PR[91] 10mm/sec CNT100;
   1:  PR[GP1:91,1] = PR[GP1:90,1] + -68.430;
   1:  PR[GP1:91,2] = PR[GP1:90,2] + 10.414;
   1:L PR[91] 10mm/sec CNT100;
   1:  PR[GP1:91,1] = PR[GP1:90,1] + -68.481;
   1:  PR[GP1:91,2] = PR[GP1:90,2] + 10.242;
   1:L PR[91] 10mm/sec CNT100;
   1:  PR[GP1:91,1] = PR[GP1:90,1] + -69.854;
   1:  PR[GP1:91,2] = PR[GP1:90,2] + 1.436;
   1:L PR[91] 10mm/sec CNT100;
   1:  PR[GP1:91,1] = PR[GP1:90,1] + -70.075;
   1:  PR[GP1:91,2] = PR[GP1:90,2] + -0.003;
   1:L PR[91] 10mm/sec CNT100;
   1:  PR[GP1:91,1] = PR[GP1:90,1] + -68.495;
   1:  PR[GP1:91,2] = PR[GP1:90,2] + -10.049;
   1:L PR[91] 10mm/sec CNT100;
   1:  PR[GP1:91,1] = PR[GP1:90,1] + -68.475;
   1:  PR[GP1:91,2] = PR[GP1:90,2] + -10.270;
   1:L PR[91] 10mm/sec CNT100;
   1:  PR[GP1:91,1] = PR[GP1:90,1] + -68.430;
   1:  PR[GP1:91,2] = PR[GP1:90,2] + -10.423;
   1:L PR[91] 10mm/sec CNT100;
   1:  PR[GP1:91,1] = PR[GP1:90,1] + -63.810;
   1:  PR[GP1:91,2] = PR[GP1:90,2] + -19.663;
   1:L PR[91] 10mm/sec CNT100;
   1:  PR[GP1:91,1] = PR[GP1:90,1] + -63.310;
   1:  PR[GP1:91,2] = PR[GP1:90,2] + -20.311;
   1:L PR[91] 10mm/sec CNT100;
   1:  PR[GP1:91,1] = PR[GP1:90,1] + -57.312;
   1:  PR[GP1:91,2] = PR[GP1:90,2] + -26.618;
   1:L PR[91] 10mm/sec CNT100;
   1:  PR[GP1:91,1] = PR[GP1:90,1] + -56.121;
   1:  PR[GP1:91,2] = PR[GP1:90,2] + -27.686;
   1:L PR[91] 10mm/sec CNT100;
   1:  PR[GP1:91,1] = PR[GP1:90,1] + -50.199;
   1:  PR[GP1:91,2] = PR[GP1:90,2] + -31.017;
   1:L PR[91] 10mm/sec CNT100;
   1:  PR[GP1:91,1] = PR[GP1:90,1] + -48.138;
   1:  PR[GP1:91,2] = PR[GP1:90,2] + -32.323;
   1:L PR[91] 10mm/sec CNT100;
   1:  PR[GP1:91,1] = PR[GP1:90,1] + -45.155;
   1:  PR[GP1:91,2] = PR[GP1:90,2] + -33.497;
   1:L PR[91] 10mm/sec CNT100;
   1:  PR[GP1:91,1] = PR[GP1:90,1] + -40.683;
   1:  PR[GP1:91,2] = PR[GP1:90,2] + -34.549;
   1:L PR[91] 10mm/sec CNT100;
   1:  PR[GP1:91,1] = PR[GP1:90,1] + -36.734;
   1:  PR[GP1:91,2] = PR[GP1:90,2] + -35.381;
   1:L PR[91] 10mm/sec CNT100;
   1:  PR[GP1:91,1] = PR[GP1:90,1] + -30.894;
   1:  PR[GP1:91,2] = PR[GP1:90,2] + -35.547;
   1:L PR[91] 10mm/sec CNT100;
   1:  PR[GP1:91,1] = PR[GP1:90,1] + -29.768;
   1:  PR[GP1:91,2] = PR[GP1:90,2] + -35.490;
   1:L PR[91] 10mm/sec CNT100;
   1:  PR[GP1:91,1] = PR[GP1:90,1] + -26.665;
   1:  PR[GP1:91,2] = PR[GP1:90,2] + -35.039;
   1:L PR[91] 10mm/sec CNT100;
   1:  PR[GP1:91,1] = PR[GP1:90,1] + -23.513;
   1:  PR[GP1:91,2] = PR[GP1:90,2] + -34.627;
   1:L PR[91] 10mm/sec CNT100;
   1:  PR[GP1:91,1] = PR[GP1:90,1] + -17.562;
   1:  PR[GP1:91,2] = PR[GP1:90,2] + -32.733;
   1:L PR[91] 10mm/sec CNT100;
   1:  PR[GP1:91,1] = PR[GP1:90,1] + -16.517;
   1:  PR[GP1:91,2] = PR[GP1:90,2] + -32.370;
   1:L PR[91] 10mm/sec CNT100;
   1:  PR[GP1:91,1] = PR[GP1:90,1] + -11.070;
   1:  PR[GP1:91,2] = PR[GP1:90,2] + -29.520;
   1:L PR[91] 10mm/sec CNT100;
   1:  PR[GP1:91,1] = PR[GP1:90,1] + -10.058;
   1:  PR[GP1:91,2] = PR[GP1:90,2] + -28.785;
   1:L PR[91] 10mm/sec CNT100;
   1:  PR[GP1:91,1] = PR[GP1:90,1] + -6.254;
   1:  PR[GP1:91,2] = PR[GP1:90,2] + -25.806;
   1:L PR[91] 10mm/sec CNT100;
   1:  PR[GP1:91,1] = PR[GP1:90,1] + -3.397;
   1:  PR[GP1:91,2] = PR[GP1:90,2] + -22.492;
   1:L PR[91] 10mm/sec CNT100;
   1:  PR[GP1:91,1] = PR[GP1:90,1] + -1.854;
   1:  PR[GP1:91,2] = PR[GP1:90,2] + -22.161;
   1:L PR[91] 10mm/sec CNT100;
   1:  PR[GP1:91,1] = PR[GP1:90,1] + 0.773;
   1:  PR[GP1:91,2] = PR[GP1:90,2] + -20.769;
   1:L PR[91] 10mm/sec CNT100;
   1:  PR[GP1:91,1] = PR[GP1:90,1] + 4.280;
   1:  PR[GP1:91,2] = PR[GP1:90,2] + -22.555;
   1:L PR[91] 10mm/sec CNT100;
   1:  PR[GP1:91,1] = PR[GP1:90,1] + 7.109;
   1:  PR[GP1:91,2] = PR[GP1:90,2] + -25.840;
   1:L PR[91] 10mm/sec CNT100;
   1:  PR[GP1:91,1] = PR[GP1:90,1] + 10.895;
   1:  PR[GP1:91,2] = PR[GP1:90,2] + -28.802;
   1:L PR[91] 10mm/sec CNT100;
   1:  PR[GP1:91,1] = PR[GP1:90,1] + 11.908;
   1:  PR[GP1:91,2] = PR[GP1:90,2] + -29.538;
   1:L PR[91] 10mm/sec CNT100;
   1:  PR[GP1:91,1] = PR[GP1:90,1] + 17.316;
   1:  PR[GP1:91,2] = PR[GP1:90,2] + -32.360;
   1:L PR[91] 10mm/sec CNT100;
   1:  PR[GP1:91,1] = PR[GP1:90,1] + 24.330;
   1:  PR[GP1:91,2] = PR[GP1:90,2] + -34.623;
   1:L PR[91] 10mm/sec CNT100;
   1:  PR[GP1:91,1] = PR[GP1:90,1] + 27.486;
   1:  PR[GP1:91,2] = PR[GP1:90,2] + -35.038;
   1:L PR[91] 10mm/sec CNT100;
   1:  PR[GP1:91,1] = PR[GP1:90,1] + 30.577;
   1:  PR[GP1:91,2] = PR[GP1:90,2] + -35.490;
   1:L PR[91] 10mm/sec CNT100;
   1:  PR[GP1:91,1] = PR[GP1:90,1] + 31.700;
   1:  PR[GP1:91,2] = PR[GP1:90,2] + -35.548;
   1:L PR[91] 10mm/sec CNT100;
   1:  PR[GP1:91,1] = PR[GP1:90,1] + 37.518;
   1:  PR[GP1:91,2] = PR[GP1:90,2] + -35.386;
   1:L PR[91] 10mm/sec CNT100;
   1:  PR[GP1:91,1] = PR[GP1:90,1] + 41.289;
   1:  PR[GP1:91,2] = PR[GP1:90,2] + -34.508;
   1:L PR[91] 10mm/sec CNT100;
   1:  PR[GP1:91,1] = PR[GP1:90,1] + 45.954;
   1:  PR[GP1:91,2] = PR[GP1:90,2] + -33.499;
   1:L PR[91] 10mm/sec CNT100;
   1:  PR[GP1:91,1] = PR[GP1:90,1] + 48.958;
   1:  PR[GP1:91,2] = PR[GP1:90,2] + -32.323;
   1:L PR[91] 10mm/sec CNT100;
   1:  PR[GP1:91,1] = PR[GP1:90,1] + 55.052;
   1:  PR[GP1:91,2] = PR[GP1:90,2] + -28.861;
   1:L PR[91] 10mm/sec CNT100;
   1:  PR[GP1:91,1] = PR[GP1:90,1] + 56.914;
   1:  PR[GP1:91,2] = PR[GP1:90,2] + -27.714;
   1:L PR[91] 10mm/sec CNT100;
   1:  PR[GP1:91,1] = PR[GP1:90,1] + 58.113;
   1:  PR[GP1:91,2] = PR[GP1:90,2] + -26.642;
   1:L PR[91] 10mm/sec CNT100;
   1:  PR[GP1:91,1] = PR[GP1:90,1] + 64.118;
   1:  PR[GP1:91,2] = PR[GP1:90,2] + -20.310;
   1:L PR[91] 10mm/sec CNT100;
   1:  PR[GP1:91,1] = PR[GP1:90,1] + 64.626;
   1:  PR[GP1:91,2] = PR[GP1:90,2] + -19.652;
   1:L PR[91] 10mm/sec CNT100;
   1:  PR[GP1:91,1] = PR[GP1:90,1] + 69.250;
   1:  PR[GP1:91,2] = PR[GP1:90,2] + -10.453;
   1:L PR[91] 10mm/sec CNT100;
   1:  PR[GP1:91,1] = PR[GP1:90,1] + 69.300;
   1:  PR[GP1:91,2] = PR[GP1:90,2] + -10.285;
   1:L PR[91] 10mm/sec CNT100;
   1:  PR[GP1:91,1] = PR[GP1:90,1] + 70.895;
   1:  PR[GP1:91,2] = PR[GP1:90,2] + -0.005;
   1:L PR[91] 10mm/sec CNT100;
   1:  PR[GP1:91,1] = PR[GP1:90,1] + 69.315;
   1:  PR[GP1:91,2] = PR[GP1:90,2] + 10.068;
   1:L PR[91] 10mm/sec CNT100;
   1:  PR[GP1:91,1] = PR[GP1:90,1] + 69.295;
   1:  PR[GP1:91,2] = PR[GP1:90,2] + 10.295;
   1:L PR[91] 10mm/sec CNT100;
   1:  PR[GP1:91,1] = PR[GP1:90,1] + 69.250;
   1:  PR[GP1:91,2] = PR[GP1:90,2] + 10.445;
   1:L PR[91] 10mm/sec CNT100;
   1:  PR[GP1:91,1] = PR[GP1:90,1] + 64.626;
   1:  PR[GP1:91,2] = PR[GP1:90,2] + 19.643;
   1:L PR[91] 10mm/sec CNT100;
   1:  PR[GP1:91,1] = PR[GP1:90,1] + 64.118;
   1:  PR[GP1:91,2] = PR[GP1:90,2] + 20.301;
   1:L PR[91] 10mm/sec CNT100;
   1:  PR[GP1:91,1] = PR[GP1:90,1] + 58.113;
   1:  PR[GP1:91,2] = PR[GP1:90,2] + 26.633;
   1:L PR[91] 10mm/sec CNT100;
   1:  PR[GP1:91,1] = PR[GP1:90,1] + 56.923;
   1:  PR[GP1:91,2] = PR[GP1:90,2] + 27.697;
   1:L PR[91] 10mm/sec CNT100;
   1:  PR[GP1:91,1] = PR[GP1:90,1] + 50.999;
   1:  PR[GP1:91,2] = PR[GP1:90,2] + 31.025;
   1:L PR[91] 10mm/sec CNT100;
   1:  PR[GP1:91,1] = PR[GP1:90,1] + 48.945;
   1:  PR[GP1:91,2] = PR[GP1:90,2] + 32.320;
   1:L PR[91] 10mm/sec CNT100;
   1:  PR[GP1:91,1] = PR[GP1:90,1] + 45.949;
   1:  PR[GP1:91,2] = PR[GP1:90,2] + 33.492;
   1:L PR[91] 10mm/sec CNT100;
   1:  PR[GP1:91,1] = PR[GP1:90,1] + 41.480;
   1:  PR[GP1:91,2] = PR[GP1:90,2] + 34.546;
   1:L PR[91] 10mm/sec CNT100;
   1:  PR[GP1:91,1] = PR[GP1:90,1] + 37.525;
   1:  PR[GP1:91,2] = PR[GP1:90,2] + 35.377;
   1:L PR[91] 10mm/sec CNT100;
   1:  PR[GP1:91,1] = PR[GP1:90,1] + 31.700;
   1:  PR[GP1:91,2] = PR[GP1:90,2] + 35.539;
   1:L PR[91] 10mm/sec CNT100;
   1:  PR[GP1:91,1] = PR[GP1:90,1] + 30.577;
   1:  PR[GP1:91,2] = PR[GP1:90,2] + 35.482;
   1:L PR[91] 10mm/sec CNT100;
   1:  PR[GP1:91,1] = PR[GP1:90,1] + 27.486;
   1:  PR[GP1:91,2] = PR[GP1:90,2] + 35.029;
   1:L PR[91] 10mm/sec CNT100;
   1:  PR[GP1:91,1] = PR[GP1:90,1] + 24.329;
   1:  PR[GP1:91,2] = PR[GP1:90,2] + 34.614;
   1:L PR[91] 10mm/sec CNT100;
   1:  PR[GP1:91,1] = PR[GP1:90,1] + 18.371;
   1:  PR[GP1:91,2] = PR[GP1:90,2] + 32.718;
   1:L PR[91] 10mm/sec CNT100;
   1:  PR[GP1:91,1] = PR[GP1:90,1] + 17.324;
   1:  PR[GP1:91,2] = PR[GP1:90,2] + 32.355;
   1:L PR[91] 10mm/sec CNT100;
   1:  PR[GP1:91,1] = PR[GP1:90,1] + 11.906;
   1:  PR[GP1:91,2] = PR[GP1:90,2] + 29.528;
   1:L PR[91] 10mm/sec CNT100;
   1:  PR[GP1:91,1] = PR[GP1:90,1] + 11.181;
   1:  PR[GP1:91,2] = PR[GP1:90,2] + 29.016;
   1:L PR[91] 10mm/sec CNT100;
   1:  PR[GP1:91,1] = PR[GP1:90,1] + 7.261;
   1:  PR[GP1:91,2] = PR[GP1:90,2] + 25.948;
   1:L PR[91] 10mm/sec CNT100;
   1:  PR[GP1:91,1] = PR[GP1:90,1] + 4.262;
   1:  PR[GP1:91,2] = PR[GP1:90,2] + 22.458;
   1:L PR[91] 10mm/sec CNT100;
   1:  PR[GP1:91,1] = PR[GP1:90,1] + 3.539;
   1:  PR[GP1:91,2] = PR[GP1:90,2] + 22.173;
   1:L PR[91] 10mm/sec CNT100;
   1:  PR[GP1:91,1] = PR[GP1:90,1] + 0.886;
   1:  PR[GP1:91,2] = PR[GP1:90,2] + 20.817;
   1:L PR[91] 10mm/sec CNT100;
   1:  PR[GP1:91,1] = PR[GP1:90,1] + -0.734;
   1:  PR[GP1:91,2] = PR[GP1:90,2] + 21.756;
   1:  PR[GP1:91,3] = PR[GP1:90,3] + 45.220;
   1:L PR[91] 10mm/sec CNT100;
   1:  PR[GP1:91,1] = PR[GP1:90,1] + -3.389;
   1:  PR[GP1:91,2] = PR[GP1:90,2] + 23.106;
   1:L PR[91] 10mm/sec CNT100;
   1:  PR[GP1:91,1] = PR[GP1:90,1] + -6.065;
   1:  PR[GP1:91,2] = PR[GP1:90,2] + 26.218;
   1:L PR[91] 10mm/sec CNT100;
   1:  PR[GP1:91,1] = PR[GP1:90,1] + -9.625;
   1:  PR[GP1:91,2] = PR[GP1:90,2] + 29.006;
   1:L PR[91] 10mm/sec CNT100;
   1:  PR[GP1:91,1] = PR[GP1:90,1] + -10.608;
   1:  PR[GP1:91,2] = PR[GP1:90,2] + 29.701;
   1:L PR[91] 10mm/sec CNT100;
   1:  PR[GP1:91,1] = PR[GP1:90,1] + -15.768;
   1:  PR[GP1:91,2] = PR[GP1:90,2] + 32.400;
   1:L PR[91] 10mm/sec CNT100;
   1:  PR[GP1:91,1] = PR[GP1:90,1] + -22.083;
   1:  PR[GP1:91,2] = PR[GP1:90,2] + 34.429;
   1:L PR[91] 10mm/sec CNT100;
   1:  PR[GP1:91,1] = PR[GP1:90,1] + -23.089;
   1:  PR[GP1:91,2] = PR[GP1:90,2] + 34.777;
   1:L PR[91] 10mm/sec CNT100;
   1:  PR[GP1:91,1] = PR[GP1:90,1] + -29.705;
   1:  PR[GP1:91,2] = PR[GP1:90,2] + 35.641;
   1:L PR[91] 10mm/sec CNT100;
   1:  PR[GP1:91,1] = PR[GP1:90,1] + -36.467;
   1:  PR[GP1:91,2] = PR[GP1:90,2] + 35.439;
   1:L PR[91] 10mm/sec CNT100;
   1:  PR[GP1:91,1] = PR[GP1:90,1] + -38.319;
   1:  PR[GP1:91,2] = PR[GP1:90,2] + 35.008;
   1:L PR[91] 10mm/sec CNT100;
   1:  PR[GP1:91,1] = PR[GP1:90,1] + -44.301;
   1:  PR[GP1:91,2] = PR[GP1:90,2] + 33.712;
   1:L PR[91] 10mm/sec CNT100;
   1:  PR[GP1:91,1] = PR[GP1:90,1] + -48.160;
   1:  PR[GP1:91,2] = PR[GP1:90,2] + 32.193;
   1:L PR[91] 10mm/sec CNT100;
   1:  PR[GP1:91,1] = PR[GP1:90,1] + -52.885;
   1:  PR[GP1:91,2] = PR[GP1:90,2] + 29.505;
   1:L PR[91] 10mm/sec CNT100;
   1:  PR[GP1:91,1] = PR[GP1:90,1] + -55.646;
   1:  PR[GP1:91,2] = PR[GP1:90,2] + 27.794;
   1:L PR[91] 10mm/sec CNT100;
   1:  PR[GP1:91,1] = PR[GP1:90,1] + -57.433;
   1:  PR[GP1:91,2] = PR[GP1:90,2] + 26.192;
   1:L PR[91] 10mm/sec CNT100;
   1:  PR[GP1:91,1] = PR[GP1:90,1] + -62.510;
   1:  PR[GP1:91,2] = PR[GP1:90,2] + 20.855;
   1:L PR[91] 10mm/sec CNT100;
   1:  PR[GP1:91,1] = PR[GP1:90,1] + -63.538;
   1:  PR[GP1:91,2] = PR[GP1:90,2] + 19.520;
   1:L PR[91] 10mm/sec CNT100;
   1:  PR[GP1:91,1] = PR[GP1:90,1] + -67.958;
   1:  PR[GP1:91,2] = PR[GP1:90,2] + 10.690;
   1:L PR[91] 10mm/sec CNT100;
   1:  PR[GP1:91,1] = PR[GP1:90,1] + -68.227;
   1:  PR[GP1:91,2] = PR[GP1:90,2] + 9.776;
   1:L PR[91] 10mm/sec CNT100;
   1:  PR[GP1:91,1] = PR[GP1:90,1] + -69.647;
   1:  PR[GP1:91,2] = PR[GP1:90,2] + 0.668;
   1:L PR[91] 10mm/sec CNT100;
   1:  PR[GP1:91,1] = PR[GP1:90,1] + -69.705;
   1:  PR[GP1:91,2] = PR[GP1:90,2] + 0.016;
   1:L PR[91] 10mm/sec CNT100;
   1:  PR[GP1:91,1] = PR[GP1:90,1] + -68.306;
   1:  PR[GP1:91,2] = PR[GP1:90,2] + -8.843;
   1:L PR[91] 10mm/sec CNT100;
   1:  PR[GP1:91,1] = PR[GP1:90,1] + -68.221;
   1:  PR[GP1:91,2] = PR[GP1:90,2] + -9.804;
   1:L PR[91] 10mm/sec CNT100;
   1:  PR[GP1:91,1] = PR[GP1:90,1] + -67.958;
   1:  PR[GP1:91,2] = PR[GP1:90,2] + -10.699;
   1:L PR[91] 10mm/sec CNT100;
   1:  PR[GP1:91,1] = PR[GP1:90,1] + -63.538;
   1:  PR[GP1:91,2] = PR[GP1:90,2] + -19.529;
   1:L PR[91] 10mm/sec CNT100;
   1:  PR[GP1:91,1] = PR[GP1:90,1] + -62.510;
   1:  PR[GP1:91,2] = PR[GP1:90,2] + -20.863;
   1:L PR[91] 10mm/sec CNT100;
   1:  PR[GP1:91,1] = PR[GP1:90,1] + -57.433;
   1:  PR[GP1:91,2] = PR[GP1:90,2] + -26.201;
   1:L PR[91] 10mm/sec CNT100;
   1:  PR[GP1:91,1] = PR[GP1:90,1] + -55.656;
   1:  PR[GP1:91,2] = PR[GP1:90,2] + -27.794;
   1:L PR[91] 10mm/sec CNT100;
   1:  PR[GP1:91,1] = PR[GP1:90,1] + -50.800;
   1:  PR[GP1:91,2] = PR[GP1:90,2] + -30.526;
   1:L PR[91] 10mm/sec CNT100;
   1:  PR[GP1:91,1] = PR[GP1:90,1] + -48.147;
   1:  PR[GP1:91,2] = PR[GP1:90,2] + -32.207;
   1:L PR[91] 10mm/sec CNT100;
   1:  PR[GP1:91,1] = PR[GP1:90,1] + -44.296;
   1:  PR[GP1:91,2] = PR[GP1:90,2] + -33.723;
   1:L PR[91] 10mm/sec CNT100;
   1:  PR[GP1:91,1] = PR[GP1:90,1] + -41.207;
   1:  PR[GP1:91,2] = PR[GP1:90,2] + -34.450;
   1:L PR[91] 10mm/sec CNT100;
   1:  PR[GP1:91,1] = PR[GP1:90,1] + -36.473;
   1:  PR[GP1:91,2] = PR[GP1:90,2] + -35.447;
   1:L PR[91] 10mm/sec CNT100;
   1:  PR[GP1:91,1] = PR[GP1:90,1] + -29.705;
   1:  PR[GP1:91,2] = PR[GP1:90,2] + -35.650;
   1:L PR[91] 10mm/sec CNT100;
   1:  PR[GP1:91,1] = PR[GP1:90,1] + -23.080;
   1:  PR[GP1:91,2] = PR[GP1:90,2] + -34.784;
   1:L PR[91] 10mm/sec CNT100;
   1:  PR[GP1:91,1] = PR[GP1:90,1] + -17.413;
   1:  PR[GP1:91,2] = PR[GP1:90,2] + -32.981;
   1:L PR[91] 10mm/sec CNT100;
   1:  PR[GP1:91,1] = PR[GP1:90,1] + -15.771;
   1:  PR[GP1:91,2] = PR[GP1:90,2] + -32.411;
   1:L PR[91] 10mm/sec CNT100;
   1:  PR[GP1:91,1] = PR[GP1:90,1] + -10.610;
   1:  PR[GP1:91,2] = PR[GP1:90,2] + -29.710;
   1:L PR[91] 10mm/sec CNT100;
   1:  PR[GP1:91,1] = PR[GP1:90,1] + -9.242;
   1:  PR[GP1:91,2] = PR[GP1:90,2] + -28.717;
   1:L PR[91] 10mm/sec CNT100;
   1:  PR[GP1:91,1] = PR[GP1:90,1] + -5.877;
   1:  PR[GP1:91,2] = PR[GP1:90,2] + -26.081;
   1:L PR[91] 10mm/sec CNT100;
   1:  PR[GP1:91,1] = PR[GP1:90,1] + -3.333;
